//Changes to the origin constraint do not affect the copy of the constraint in the instance of the DynamicConstraint_Container.
//For this reason, the container is being refreshed here							
fbDynConstraintContainer.Clear();
fbDynConstraintContainer.AddConstraint(fbDynConstraintPath);
fbDynConstraintContainer.AddConstraint(fbDynConstraintCoordinates);
END_METHOD

METHOD SetDynConstraint_C : BOOL //Dynamic constraints for individual coordinates.
VAR_INPUT
    V : MC_LREAL; //equivalent to data type LREAL + MC_DEFAULT, MC_MAXIMUM
    A : MC_LREAL; //equivalent to data type LREAL + MC_DEFAULT, MC_MAXIMUM
    D : MC_LREAL; //equivalent to data type LREAL + MC_DEFAULT, MC_MAXIMUM
    J : MC_LREAL; //equivalent to data type LREAL + MC_DEFAULT, MC_MAXIMUM
END_VAR
THIS^.fbDynConstraintCoordinates.SetLimit(	Coordinate := Coord_Mcs_C1, 
											V := V, 
											A := A, 
											D := D, 
											J := J);											

//Changes to the origin constraint do not affect the copy of the constraint in the instance of the DynamicConstraint_Container.
//For this reason, the container is being refreshed here							
fbDynConstraintContainer.Clear();
fbDynConstraintContainer.AddConstraint(fbDynConstraintPath);
fbDynConstraintContainer.AddConstraint(fbDynConstraintCoordinates);
END_METHOD

METHOD SetDynConstraint_Path : BOOL //One dimensional dynamic constraint along the XY-components of a path, ignoring non-tangential effects.
VAR_INPUT
    V : MC_LREAL; //equivalent to data type LREAL + MC_DEFAULT, MC_MAXIMUM
    A : MC_LREAL; //equivalent to data type LREAL + MC_DEFAULT, MC_MAXIMUM
    D : MC_LREAL; //equivalent to data type LREAL + MC_DEFAULT, MC_MAXIMUM
    J : MC_LREAL; //equivalent to data type LREAL + MC_DEFAULT, MC_MAXIMUM
END_VAR
THIS^.fbDynConstraintPath.SetValuesVADJ(V := V, 
										A := A, 
										D := D, 
										J := J);											

//Changes to the origin constraint do not affect the copy of the constraint in the instance of the DynamicConstraint_Container.
//For this reason, the container is being refreshed here							
fbDynConstraintContainer.Clear();
fbDynConstraintContainer.AddConstraint(fbDynConstraintPath);
fbDynConstraintContainer.AddConstraint(fbDynConstraintCoordinates);
END_METHOD

METHOD SetDynConstraint_X : BOOL //Dynamic constraints for individual coordinates.
VAR_INPUT
    V : MC_LREAL; //equivalent to data type LREAL + MC_DEFAULT, MC_MAXIMUM
    A : MC_LREAL; //equivalent to data type LREAL + MC_DEFAULT, MC_MAXIMUM
    D : MC_LREAL; //equivalent to data type LREAL + MC_DEFAULT, MC_MAXIMUM
    J : MC_LREAL; //equivalent to data type LREAL + MC_DEFAULT, MC_MAXIMUM
END_VAR
THIS^.fbDynConstraintCoordinates.SetLimit(	Coordinate := Coord_Mcs_X, 
											V := V, 
											A := A, 
											D := D, 
											J := J);											

//Changes to the origin constraint do not affect the copy of the constraint in the instance of the DynamicConstraint_Container.
//For this reason, the container is being refreshed here							
fbDynConstraintContainer.Clear();
fbDynConstraintContainer.AddConstraint(fbDynConstraintPath);
fbDynConstraintContainer.AddConstraint(fbDynConstraintCoordinates);
END_METHOD

METHOD SetDynConstraint_Y : BOOL //Dynamic constraints for individual coordinates.
VAR_INPUT
    V : MC_LREAL; //equivalent to data type LREAL + MC_DEFAULT, MC_MAXIMUM
    A : MC_LREAL; //equivalent to data type LREAL + MC_DEFAULT, MC_MAXIMUM
    D : MC_LREAL; //equivalent to data type LREAL + MC_DEFAULT, MC_MAXIMUM
    J : MC_LREAL; //equivalent to data type LREAL + MC_DEFAULT, MC_MAXIMUM
END_VAR
THIS^.fbDynConstraintCoordinates.SetLimit(	Coordinate := Coord_Mcs_Y, 
											V := V, 
											A := A, 
											D := D, 
											J := J);											

//Changes to the origin constraint do not affect the copy of the constraint in the instance of the DynamicConstraint_Container.
//For this reason, the container is being refreshed here							
fbDynConstraintContainer.Clear();
fbDynConstraintContainer.AddConstraint(fbDynConstraintPath);
fbDynConstraintContainer.AddConstraint(fbDynConstraintCoordinates);
END_METHOD

METHOD SetDynConstraint_Z : BOOL //Dynamic constraints for individual coordinates.
VAR_INPUT
    V : MC_LREAL; //equivalent to data type LREAL + MC_DEFAULT, MC_MAXIMUM
    A : MC_LREAL; //equivalent to data type LREAL + MC_DEFAULT, MC_MAXIMUM
    D : MC_LREAL; //equivalent to data type LREAL + MC_DEFAULT, MC_MAXIMUM
    J : MC_LREAL; //equivalent to data type LREAL + MC_DEFAULT, MC_MAXIMUM
END_VAR
THIS^.fbDynConstraintCoordinates.SetLimit(	Coordinate := Coord_Mcs_Z, 
											V := MC_DEFAULT, 
											A := A, 
											D := D, 
											J := J);											

//Changes to the origin constraint do not affect the copy of the constraint in the instance of the DynamicConstraint_Container.
//For this reason, the container is being refreshed here							
fbDynConstraintContainer.Clear();
fbDynConstraintContainer.AddConstraint(fbDynConstraintPath);
fbDynConstraintContainer.AddConstraint(fbDynConstraintCoordinates);
END_METHOD

METHOD SetRouteToParent : HRESULT
VAR_INPUT
	ipRoute : I_CH_LIST;
END_VAR
IF ipRoute = 0 THEN
	//Clear on empty input
	THIS^.fbRouteRemaining.Clear();
	THIS^.fbRouteComplete.Clear();
ELSE	
	//set as new route
	THIS^.fbRouteRemaining.Duplicate(ipRoute);
	THIS^.fbRouteComplete.Duplicate(ipRoute);	
END_IF
END_METHOD

{attribute 'monitoring':='call'}
(* Velocity is zero *)
PROPERTY Standstill : BOOL
GET
Standstill := TRUE;
Standstill := Standstill AND THIS^.PlanarMover.MCTOPLC.SET.SetVelo.x = 0;
Standstill := Standstill AND THIS^.PlanarMover.MCTOPLC.SET.SetVelo.y = 0;
Standstill := Standstill AND THIS^.PlanarMover.MCTOPLC.SET.SetVelo.z = 0;
Standstill := Standstill AND THIS^.PlanarMover.MCTOPLC.SET.SetVelo.a = 0;
Standstill := Standstill AND THIS^.PlanarMover.MCTOPLC.SET.SetVelo.b = 0;
Standstill := Standstill AND THIS^.PlanarMover.MCTOPLC.SET.SetVelo.c = 0;
END_GET
END_PROPERTY

METHOD StartExternalSetpoint : HRESULT
THIS^.eActiveCommand 				:= CHALET_NC.E_NcAxisCommands.StartExternalSetpoint;
THIS^.fbFeedback.ActiveCommand 		:= TO_STRING(THIS^.eActiveCommand);		
THIS^.fbFeedback.Busy 				:= TRUE;


IF THIS^.fbMover.MCTOPLC.STD.State <> MC_PLANAR_STATE.Enabled THEN
	//Error wrong state
	
	;//zzz Todo Error message

ELSIF THIS^.bFeedExternalSetpointActive AND THIS^.nSeqStartExternalSetpoint = 999 THEN
	//Do nothing, setpoint is already active	
	THIS^.fbFeedbackExternalSetpointStartSeq.Done		:= TRUE;
	
ELSE
	
	//Start of internal sequence
	THIS^.fbFeedbackExternalSetpointStartSeq.Busy		:= TRUE;
	THIS^.nSeqStartExternalSetpoint := 1;
END_IF



StartExternalSetpoint := S_OK;
END_METHOD

METHOD StopExternalSetpoint : HRESULT
VAR_INPUT
END_VAR
AxisSetpointX.PowerOff();
AxisSetpointY.PowerOff();
AxisSetpointZ.PowerOff();
AxisSetpointA.PowerOff();
AxisSetpointB.PowerOff();
AxisSetpointC.PowerOff();


THIS^.eActiveCommand 				:= CHALET_NC.E_NcAxisCommands.StopExternalSetpoint;
THIS^.fbFeedback.ActiveCommand 		:= TO_STRING(THIS^.eActiveCommand);	
THIS^.fbFeedback.LastCommandAccepted:= TRUE;		


//Reset some flags
THIS^.nSeqStartExternalSetpoint := 0;
THIS^.bEvaluateFeedback := FALSE;
THIS^.ipMasterMover := 0;

IF THIS^.bFeedExternalSetpointActive THEN
	THIS^.fbMover.StopExternalSetpointGeneration(THIS^.fbFeedbackExtStop);	
	THIS^.bFeedExternalSetpointActive 	:= FALSE;
	THIS^.fbFeedback.Busy 				:= TRUE;
ELSE
	THIS^.fbFeedback.Done 				:= TRUE;
END_IF


StopExternalSetpoint := S_OK;
END_METHOD

{attribute 'monitoring':='call'}
//Interface to CHALET system to which this object belongs
PROPERTY System : I_XP_System_PLC
GET
//get I_x_System_PLC interface from I_x_System_Registration
__QUERYINTERFACE(THIS^.ipXpSystem, System);
END_GET
END_PROPERTY

{attribute 'monitoring':='call'}
PROPERTY TargetStation : STRING
GET
TargetStation := THIS^.sTargetStation;
END_GET
SET
THIS^.sTargetStation := TargetStation;
END_SET
END_PROPERTY

METHOD PUBLIC Update : HRESULT
VAR
	ipObject : I_CH_Object;
END_VAR

VAR_INST
	{attribute 'hide'}
	fbCmdNotPossibleCollision : FB_TcAlarm;
	{attribute 'hide'}
	nFeedbackOidOld : UDINT;
	{attribute 'hide'}	
	nOldNcErrorCode 		: UDINT;
	{attribute 'hide'}	
	fbAlarmNcErrorCode		: FB_TcAlarm;
END_VAR
THIS^.Prepare();//Prepare time-critical information, if not already done

THIS^.UpdateExternalSetpoint();
THIS^.UpdateUnknownLevel();

// ********************** Set feedback depending on active command *******************************
CASE THIS^.eActiveCommand OF
	E_NcAxisCommands.None: 
		//Display if a Mover Error is active during no command is active
		IF THIS^.fbMover.Error AND NOT fbFeedback.Error THEN 
			IF THIS^.fbMover.ErrorId <> 1810(*ignore ADSERR_DEVICE_INVALIDSTATE*) THEN
				fbFeedback.ErrorId 			:= THIS^.fbMover.ErrorID;
				fbFeedback.ActiveCommand 	:= TO_STRING(E_NcAxisCommands.None);	
				fbFeedback.ClearObjectInfo();
			END_IF
		END_IF

	E_NcAxisCommands.Initialize:
		fbFeedback.Busy 			:= NOT THIS^.bInitDone;
		fbFeedback.Done 			:= THIS^.bInitDone;
		fbFeedback.ErrorId 			:= 0;
		fbFeedback.ClearObjectInfo();
		                        	
	E_NcAxisCommands.MoveA:     	
		fbFeedback.Busy 			:= fbFeedbackMoveA.Busy;
		fbFeedback.Done 			:= fbFeedbackMoveA.Done;
		fbFeedback.ErrorId 			:= fbFeedbackMoveA.ErrorID;
        fbFeedback.ObjectInfo		:= fbFeedbackMoveA.objectInfo;
                                	
	E_NcAxisCommands.MoveB:     	
		fbFeedback.Busy 			:= fbFeedbackMoveB.Busy;
		fbFeedback.Done 			:= fbFeedbackMoveB.Done;
		fbFeedback.ErrorId 			:= fbFeedbackMoveB.ErrorID;
        fbFeedback.ObjectInfo		:= fbFeedbackMoveB.objectInfo;
                                	
	E_NcAxisCommands.MoveC:     	
		fbFeedback.Busy 			:= fbFeedbackMoveC.Busy;
		fbFeedback.Done 			:= fbFeedbackMoveC.Done;
		fbFeedback.ErrorId 			:= fbFeedbackMoveC.ErrorID;
        fbFeedback.ObjectInfo		:= fbFeedbackMoveC.objectInfo;
                                	
	E_NcAxisCommands.MoveXY:    	
		fbFeedback.Busy 			:= fbFeedbackMoveXY.Busy;
		fbFeedback.Done 			:= fbFeedbackMoveXY.Done;
		fbFeedback.ErrorId 			:= fbFeedbackMoveXY.ErrorID;
        fbFeedback.ObjectInfo		:= fbFeedbackMoveXY.objectInfo;
                                	
	E_NcAxisCommands.MoveZ:     	
		fbFeedback.Busy 			:= fbFeedbackMoveZ.Busy;
		fbFeedback.Done 			:= fbFeedbackMoveZ.Done;
		fbFeedback.ErrorId 			:= fbFeedbackMoveZ.ErrorID;
        fbFeedback.ObjectInfo		:= fbFeedbackMoveZ.objectInfo;
                                	
	E_NcAxisCommands.Enable:    	
		fbFeedback.Busy 			:= fbFeedbackEnable.Busy;
		fbFeedback.Done 			:= fbFeedbackEnable.Done;
		fbFeedback.ErrorId 			:= fbFeedbackEnable.ErrorID;
        fbFeedback.ObjectInfo		:= fbFeedbackEnable.objectInfo;
                                	
	E_NcAxisCommands.Disable:   	
		fbFeedback.Busy 			:= fbFeedbackDisable.Busy;
		fbFeedback.Done 			:= fbFeedbackDisable.Done;
		fbFeedback.ErrorId 			:= fbFeedbackDisable.ErrorID;
        fbFeedback.ObjectInfo		:= fbFeedbackDisable.objectInfo;
                                	
	E_NcAxisCommands.Reset:     	
		fbFeedback.Busy 			:= fbFeedbackReset.Busy;
		fbFeedback.Done 			:= fbFeedbackReset.Done;
		fbFeedback.ErrorId 			:= fbFeedbackReset.ErrorID;
        fbFeedback.ObjectInfo		:= fbFeedbackReset.objectInfo;
                                	
	E_NcAxisCommands.Halt:      	
		fbFeedback.Busy 			:= fbFeedbackHalt.Busy;
		fbFeedback.Done 			:= fbFeedbackHalt.Done;
		fbFeedback.ErrorId 			:= fbFeedbackHalt.ErrorID;
        fbFeedback.ObjectInfo		:= fbFeedbackHalt.objectInfo;

	E_NcAxisCommands.AddToGroupe:
		fbFeedback.Busy 			:= fbFeedbackAddToGrp.Busy;
		fbFeedback.Done 			:= fbFeedbackAddToGrp.Done;
		fbFeedback.ErrorId 			:= fbFeedbackAddToGrp.ErrorID;
        fbFeedback.ObjectInfo		:= fbFeedbackAddToGrp.objectInfo;

	E_NcAxisCommands.RemoveFromGroupe:
		fbFeedback.Busy 			:= fbFeedbackRmvFromGrp.Busy;
		fbFeedback.Done 			:= fbFeedbackRmvFromGrp.Done;
		fbFeedback.ErrorId 			:= fbFeedbackRmvFromGrp.ErrorID;
        fbFeedback.ObjectInfo		:= fbFeedbackRmvFromGrp.objectInfo;
		
	E_NcAxisCommands.JoinTrack:
		fbFeedback.Busy 			:= fbFeedbackJoinTrack.Busy;
		fbFeedback.Done 			:= fbFeedbackJoinTrack.Done;
		fbFeedback.ErrorId 			:= fbFeedbackJoinTrack.ErrorID;
        fbFeedback.ObjectInfo		:= fbFeedbackJoinTrack.objectInfo;
		
	E_NcAxisCommands.MoveOnTrack:
		fbFeedback.Busy 			:= fbFeedbackMoveOnTrack.Busy;
		fbFeedback.Done 			:= fbFeedbackMoveOnTrack.Done;
		fbFeedback.ErrorId 			:= fbFeedbackMoveOnTrack.ErrorID;
        fbFeedback.ObjectInfo		:= fbFeedbackMoveOnTrack.objectInfo;
		
			
	E_NcAxisCommands.StartExternalSetpoint:
		;// in Subroutine "UpdateExternalSetpoint"
	
	E_NcAxisCommands.StopExternalSetpoint:
		;// in Subroutine "UpdateExternalSetpoint"		
			
	E_NcAxisCommands.LiftFromUnknownLevel:
		fbFeedback.Busy 			:= fbFeedbackLiftFromUnknown.Busy;
		fbFeedback.Done 			:= fbFeedbackLiftFromUnknown.Done;
		fbFeedback.ErrorId 			:= fbFeedbackLiftFromUnknown.ErrorID;
        fbFeedback.ClearObjectInfo();
	
	E_NcAxisCommands.LowerToUnknownLevel:
		fbFeedback.Busy 			:= fbFeedbackLowerToUnknown.Busy;
		fbFeedback.Done 			:= fbFeedbackLowerToUnknown.Done;
		fbFeedback.ErrorId 			:= fbFeedbackLowerToUnknown.ErrorID;
        fbFeedback.ClearObjectInfo();
		
	ELSE//External command in subclass
		;
END_CASE


// **********************  Stop to execute commands on .done or .error ***************************
IF fbFeedback.Done OR THIS^.fbFeedback.Error THEN
	eActiveCommand 				:= E_NcAxisCommands.None;
END_IF


// **********************  Get interface to Feedback.ObjectInfo ***************************
IF Feedback.ObjectInfoEx.Id <> 0 AND Feedback.ObjectInfoEx.Id <> nFeedbackOidOld THEN
	CASE Feedback.ObjectInfo.ObjectType OF
		EPlanarObjectType.Mover:
			Feedback.ObjectInfoEx.ipObject := THIS^.ipXPSystem.MoversPresent.FindOID(Feedback.ObjectInfo.Id);
			
		EPlanarObjectType.Track:
				Feedback.ObjectInfoEx.ipObject := THIS^.ipXPSystem.Tracks.FindOID(Feedback.ObjectInfo.Id);
		
		EPlanarObjectType.Environment:
				Feedback.ObjectInfoEx.ipObject := THIS^.ipXPSystem.Enviroment;
				
		ELSE 
			Feedback.ObjectInfoEx.ipObject := 0;
	END_CASE
END_IF
nFeedbackOidOld := Feedback.ObjectInfo.Id;



// **********************  Write NC-Error(Mover.MCTOPLC.ErrorCode) in TC3 Eventlogger ***************************
IF (THIS^.fbMover.MCTOPLC.STD.ErrorCode = 0 AND fbAlarmNcErrorCode.bRaised) THEN
	//No error - Reset	
	fbAlarmNcErrorCode.Clear(0,0);
	
ELSIF (THIS^.fbMover.MCTOPLC.STD.ErrorCode = 0) THEN
	; //Nothing
	
ELSIF (nOldNcErrorCode <> THIS^.fbMover.MCTOPLC.STD.ErrorCode) THEN
	//New Error - Reset, Create and Raise
	fbAlarmNcErrorCode.Clear(0,0);
	fbAlarmNcErrorCode.Create(	eventClass		:= TC_EVENT_CLASSES.Tc3_NcErrorCodes, 
								nEventId		:= (TO_DWORD(THIS^.fbMover.MCTOPLC.STD.ErrorCode) AND 16#FFFF), //Cut HRESULT to 4 digit error code
								eSeverity		:= TcEventSeverity.Error, 
								ipSourceInfo 	:= THIS^.fbSourceInfo, 
								bWithConfirmation := FALSE);
	fbAlarmNcErrorCode.ipArguments.Clear();
	fbAlarmNcErrorCode.Raise(0);
ELSE
	//Alarm is already active
	;
END_IF
nOldNcErrorCode := THIS^.fbMover.MCTOPLC.STD.ErrorCode;



// **********************  Raise alarm on collision error ***************************
ipObject := THIS^.fbFeedback.ObjectInfoEx.ipObject;
IF THIS^.fbFeedback.Error AND (ipObject <> 0) AND NOT fbCmdNotPossibleCollision.bRaised THEN
	fbCmdNotPossibleCollision.CreateEx(stEventEntry := TC_EVENTS.CHALET_XPlanar_Events.CommandNotPossibleCollision, bWithConfirmation := FALSE, ipSourceInfo := THIS^.fbSourceInfo);
	//Command "{1}" not possible. Possible collision with "{2}"
	fbCmdNotPossibleCollision.ipArguments.AddStringByValue(THIS^.fbFeedback.ActiveCommand).AddStringByValue(ipObject.LUID);
	fbCmdNotPossibleCollision.Raise(0);
ELSIF NOT THIS^.fbFeedback.Error OR ipObject = 0 THEN
	fbCmdNotPossibleCollision.Clear(0,0);	
END_IF




//Update xplanar object
THIS^.fbMover.Update();



//Update feedback object
fbFeedbackMoveA.Update(); 
fbFeedbackMoveB.Update(); 
fbFeedbackMoveC.Update(); 
fbFeedbackMoveXY.Update(); 
fbFeedbackMoveZ.Update(); 
fbFeedbackEnable.Update(); 
fbFeedbackDisable.Update(); 
fbFeedbackReset.Update(); 
fbFeedbackAddToGrp.Update(); 
fbFeedbackRmvFromGrp.Update(); 
fbFeedbackHalt.Update(); 
fbFeedbackJoinTrack.Update(); 
fbFeedbackMoveOnTrack.Update();
END_METHOD

METHOD PROTECTED UpdateExternalSetpoint : HRESULT
VAR
	SetPos, SetVelo, SetAcc : MoverVector;
	hr : HRESULT;
	stStartOptions : ST_ExternalSetpointGenerationOptions;
	stPosDifferenceToMasterMover : MoverVector;
	stPosOffsetMasterMover : MoverVector;
	stVeloOffsetMasterMover : MoverVector;
	stAccOffsetMasterMover : MoverVector;
END_VAR
IF NOT THIS^.Enabled THEN
	THIS^.nSeqStartExternalSetpoint := 0;
	THIS^.bFeedExternalSetpointActive := FALSE;
	THIS^.bEvaluateFeedback := FALSE;
END_IF


CASE nSeqStartExternalSetpoint OF
	0: //Wait for start
		;
		
	1: 	//store position of Master-Mover
		IF (THIS^.ipMasterMover <> 0) THEN
			THIS^.stMasterPositionAtStart := THIS^.ipMasterMover.PositionSet;
		END_IF

		//Reset all axis
		IF AxisSetpointX.Mapped THEN
			AxisSetpointX.Reset();
		END_IF
		IF AxisSetpointY.Mapped THEN
			AxisSetpointY.Reset();
		END_IF
		IF AxisSetpointZ.Mapped THEN
			AxisSetpointZ.Reset();
		END_IF
		IF AxisSetpointA.Mapped THEN
			AxisSetpointA.Reset();
		END_IF
		IF AxisSetpointB.Mapped THEN
			AxisSetpointB.Reset();
		END_IF
		IF AxisSetpointC.Mapped THEN
			AxisSetpointC.Reset();
		END_IF
		nSeqStartExternalSetpoint := nSeqStartExternalSetpoint + 1;		
		
		
	2: //Wait for feedback
		IF AxisSetpointX.Mapped THEN hr := GetMostSignificant(hr, AxisSetpointX.Feedback.HR); END_IF
		IF AxisSetpointY.Mapped THEN hr := GetMostSignificant(hr, AxisSetpointY.Feedback.HR); END_IF
		IF AxisSetpointZ.Mapped THEN hr := GetMostSignificant(hr, AxisSetpointZ.Feedback.HR); END_IF
		IF AxisSetpointA.Mapped THEN hr := GetMostSignificant(hr, AxisSetpointA.Feedback.HR); END_IF
		IF AxisSetpointB.Mapped THEN hr := GetMostSignificant(hr, AxisSetpointB.Feedback.HR); END_IF
		IF AxisSetpointC.Mapped THEN hr := GetMostSignificant(hr, AxisSetpointC.Feedback.HR); END_IF	
		IF hr = S_OK THEN
		 	nSeqStartExternalSetpoint := nSeqStartExternalSetpoint + 1;	
		END_IF
		
	3: 	//Reset all axis
		IF AxisSetpointX.Mapped THEN
			AxisSetpointX.PowerOn();
		END_IF
		IF AxisSetpointY.Mapped THEN
			AxisSetpointY.PowerOn();
		END_IF
		IF AxisSetpointZ.Mapped THEN
			AxisSetpointZ.PowerOn();
		END_IF
		IF AxisSetpointA.Mapped THEN
			AxisSetpointA.PowerOn();
		END_IF
		IF AxisSetpointB.Mapped THEN
			AxisSetpointB.PowerOn();
		END_IF
		IF AxisSetpointC.Mapped THEN
			AxisSetpointC.PowerOn();
		END_IF
		nSeqStartExternalSetpoint := nSeqStartExternalSetpoint + 1;		
		
	4: //Wait for feedback
		IF AxisSetpointX.Mapped THEN hr := GetMostSignificant(hr, AxisSetpointX.Feedback.HR); END_IF
		IF AxisSetpointY.Mapped THEN hr := GetMostSignificant(hr, AxisSetpointY.Feedback.HR); END_IF
		IF AxisSetpointZ.Mapped THEN hr := GetMostSignificant(hr, AxisSetpointZ.Feedback.HR); END_IF
		IF AxisSetpointA.Mapped THEN hr := GetMostSignificant(hr, AxisSetpointA.Feedback.HR); END_IF
		IF AxisSetpointB.Mapped THEN hr := GetMostSignificant(hr, AxisSetpointB.Feedback.HR); END_IF
		IF AxisSetpointC.Mapped THEN hr := GetMostSignificant(hr, AxisSetpointC.Feedback.HR); END_IF	
		IF hr = S_OK THEN
		 	nSeqStartExternalSetpoint := nSeqStartExternalSetpoint + 1;	
		END_IF

	5: 	//Enable all axis
		IF AxisSetpointX.Mapped THEN
			AxisSetpointX.SetActPosition(0.0);
		END_IF
		IF AxisSetpointY.Mapped THEN
			AxisSetpointY.SetActPosition(0.0);
		END_IF
		IF AxisSetpointZ.Mapped THEN
			AxisSetpointZ.SetActPosition(0.0);
		END_IF
		IF AxisSetpointA.Mapped THEN
			AxisSetpointA.SetActPosition(0.0);
		END_IF
		IF AxisSetpointB.Mapped THEN
			AxisSetpointB.SetActPosition(0.0);
		END_IF
		IF AxisSetpointC.Mapped THEN
			AxisSetpointC.SetActPosition(0.0);
		END_IF
		nSeqStartExternalSetpoint := nSeqStartExternalSetpoint + 1;		
		
	6: //Wait for feedback
		IF AxisSetpointX.Mapped THEN hr := GetMostSignificant(hr, AxisSetpointX.Feedback.HR); END_IF
		IF AxisSetpointY.Mapped THEN hr := GetMostSignificant(hr, AxisSetpointY.Feedback.HR); END_IF
		IF AxisSetpointZ.Mapped THEN hr := GetMostSignificant(hr, AxisSetpointZ.Feedback.HR); END_IF
		IF AxisSetpointA.Mapped THEN hr := GetMostSignificant(hr, AxisSetpointA.Feedback.HR); END_IF
		IF AxisSetpointB.Mapped THEN hr := GetMostSignificant(hr, AxisSetpointB.Feedback.HR); END_IF
		IF AxisSetpointC.Mapped THEN hr := GetMostSignificant(hr, AxisSetpointC.Feedback.HR); END_IF	
		IF hr = S_OK THEN
		 	nSeqStartExternalSetpoint := nSeqStartExternalSetpoint + 1;	
		END_IF

		
	7: // Activate external setpoint mode on mover
		stStartOptions.Mode := MC_EXTERNAL_SET_POSITION_MODE.Relative;
		THIS^.fbMover.StartExternalSetpointGeneration(	commandFeedback	:= THIS^.fbFeedbackExtStart,
														options 		:= stStartOptions);
		THIS^.bFeedExternalSetpointActive := TRUE;												
		nSeqStartExternalSetpoint := nSeqStartExternalSetpoint + 1;
	
		
	8: 
		THIS^.bEvaluateFeedback := TRUE;
		IF THIS^.fbFeedbackExtStart.Done THEN
			//Finish Sequence
			fbFeedbackExternalSetpointStartSeq.Done := TRUE;
			nSeqStartExternalSetpoint := 999;
		END_IF
		
	999: // finish seqence feedback
		
		
	1000..1999:
		//Error
		fbFeedbackExternalSetpointStartSeq.HR := E_FAIL;
END_CASE



IF THIS^.bFeedExternalSetpointActive THEN
	SetPos.X := AxisSetpointX.SetPosition;
	SetPos.Y := AxisSetpointY.SetPosition;
	SetPos.Z := AxisSetpointZ.SetPosition;
	SetPos.A := AxisSetpointA.SetPosition;
	SetPos.B := AxisSetpointB.SetPosition;
	SetPos.C := AxisSetpointC.SetPosition;
	
	SetVelo.X := AxisSetpointX.SetVelocity;
	SetVelo.Y := AxisSetpointY.SetVelocity;
	SetVelo.Z := AxisSetpointZ.SetVelocity;
	SetVelo.A := AxisSetpointA.SetVelocity;
	SetVelo.B := AxisSetpointB.SetVelocity;
	SetVelo.C := AxisSetpointC.SetVelocity;
	
	SetAcc.X := AxisSetpointX.SetAcceleration;
	SetAcc.Y := AxisSetpointY.SetAcceleration;
	SetAcc.Z := AxisSetpointZ.SetAcceleration;
	SetAcc.A := AxisSetpointA.SetAcceleration;
	SetAcc.B := AxisSetpointB.SetAcceleration;
	SetAcc.C := AxisSetpointC.SetAcceleration;
	
	IF THIS^.ipMasterMover <> 0 THEN
		//Difference to gearIn position
		stPosDifferenceToMasterMover := F_Vector_Subtraction(	minuend := THIS^.ipMasterMover.PositionSet, 
																subtrahend := stMasterPositionAtStart);
		//Add scaling factor	
		stPosOffsetMasterMover := F_Vector_Multiplication(	factor1 := stPosDifferenceToMasterMover,
															factor2 := THIS^.stMasterMovementScaling);							
		stVeloOffsetMasterMover := F_Vector_Multiplication(	factor1 := THIS^.ipMasterMover.VelocitySet,
															factor2 := THIS^.stMasterMovementScaling);							
		stAccOffsetMasterMover := F_Vector_Multiplication(	factor1 := THIS^.ipMasterMover.AccelerationSet,
															factor2 := THIS^.stMasterMovementScaling);						
		
		
		//Add Mastermover-Offest to 6-Axis-Offset
		SetPos := F_Vector_Addition( 	summand1 := stPosOffsetMasterMover,
									 	summand2 := SetPos);
		SetVelo := F_Vector_Addition( 	summand1 := stVeloOffsetMasterMover,
									 	summand2 := SetVelo);
		SetAcc := F_Vector_Addition( 	summand1 := stAccOffsetMasterMover,
									 	summand2 := SetAcc);
														
	END_IF
	
	//Send data to mover
	THIS^.fbMover.SetExternalSetpoint(	setPosition 		:= SetPos, 
										setVelocity 		:= SetVelo,
										setAcceleration 	:= SetAcc);
END_IF



CASE THIS^.eActiveCommand OF
	//Add the 6 axis to the feedback			
	E_NcAxisCommands.StartExternalSetpoint:
		//Only check MC_PlanarFeedback if cmd is active. Ignore old feedback
		IF THIS^.bEvaluateFeedback THEN
			fbFeedback.Busy 		:= fbFeedbackExtStart.Busy;
			fbFeedback.Done 		:= fbFeedbackExtStart.Done;
			fbFeedback.ErrorId 		:= fbFeedbackExtStart.ErrorID;
			fbFeedback.ClearObjectInfo();
		END_IF
		fbFeedback.HR := GetMostSignificant(fbFeedback.HR, fbFeedbackExternalSetpointStartSeq.HR);
		IF AxisSetpointX.Mapped THEN fbFeedback.HR := GetMostSignificant(fbFeedback.HR, AxisSetpointX.Feedback.HR);END_IF
		IF AxisSetpointY.Mapped THEN fbFeedback.HR := GetMostSignificant(fbFeedback.HR, AxisSetpointY.Feedback.HR);END_IF
		IF AxisSetpointZ.Mapped THEN fbFeedback.HR := GetMostSignificant(fbFeedback.HR, AxisSetpointZ.Feedback.HR);END_IF
		IF AxisSetpointA.Mapped THEN fbFeedback.HR := GetMostSignificant(fbFeedback.HR, AxisSetpointA.Feedback.HR);END_IF
		IF AxisSetpointB.Mapped THEN fbFeedback.HR := GetMostSignificant(fbFeedback.HR, AxisSetpointB.Feedback.HR);END_IF
		IF AxisSetpointC.Mapped THEN fbFeedback.HR := GetMostSignificant(fbFeedback.HR, AxisSetpointC.Feedback.HR);END_IF
		
	//Add the 6 axis to the feedback	
	E_NcAxisCommands.StopExternalSetpoint:
		fbFeedback.Busy 		:= fbFeedbackExtStop.Busy;
		fbFeedback.Done 		:= fbFeedbackExtStop.Done;
		fbFeedback.ErrorId 		:= fbFeedbackExtStop.ErrorID;
		fbFeedback.ClearObjectInfo(); 
		IF AxisSetpointX.Mapped THEN fbFeedback.HR := GetMostSignificant(fbFeedback.HR, AxisSetpointX.Feedback.HR);END_IF
		IF AxisSetpointY.Mapped THEN fbFeedback.HR := GetMostSignificant(fbFeedback.HR, AxisSetpointY.Feedback.HR);END_IF
		IF AxisSetpointZ.Mapped THEN fbFeedback.HR := GetMostSignificant(fbFeedback.HR, AxisSetpointZ.Feedback.HR);END_IF
		IF AxisSetpointA.Mapped THEN fbFeedback.HR := GetMostSignificant(fbFeedback.HR, AxisSetpointA.Feedback.HR);END_IF
		IF AxisSetpointB.Mapped THEN fbFeedback.HR := GetMostSignificant(fbFeedback.HR, AxisSetpointB.Feedback.HR);END_IF
		IF AxisSetpointC.Mapped THEN fbFeedback.HR := GetMostSignificant(fbFeedback.HR, AxisSetpointC.Feedback.HR);END_IF
END_CASE		


fbFeedbackExtStart.Update(); 
fbFeedbackExtStop.Update(); 


IF AxisSetpointX.Mapped THEN AxisSetpointX.Update() ;END_IF
IF AxisSetpointY.Mapped THEN AxisSetpointY.Update() ;END_IF
IF AxisSetpointZ.Mapped THEN AxisSetpointZ.Update() ;END_IF
IF AxisSetpointA.Mapped THEN AxisSetpointA.Update() ;END_IF
IF AxisSetpointB.Mapped THEN AxisSetpointB.Update() ;END_IF
IF AxisSetpointC.Mapped THEN AxisSetpointC.Update() ;END_IF
END_METHOD

METHOD PROTECTED UpdateUnknownLevel : HRESULT
VAR
	hr : HRESULT;
	stForceLimitMax: Tc3_XPlanarUtility.Force6D;
	stForceLimitMin: Tc3_XPlanarUtility.Force6D;
	stPosLagValueTemp : MoverVector;
	ipComObject: Tc3_Module.ITComObject;
	pstForcesAtBeginn : POINTER TO MoverVector;
END_VAR
VAR_INST
	fLowerNPerS : LREAL := 30.0;
	fLiftNPerS : LREAL := 50.0;
	fMaxForceFactor : LREAL := 1.0;
	fMinForceFactor : LREAL := 0.1;
	fPowerFactor : LREAL := 1.0;
	fCycleTime_s : LREAL; //[s]	
	bDoOnceIfDisabled : BOOL;
	stLagValuesAtBeginn : MoverVector;
	stForcesAtBeginn :  MoverVector;
	stForceLimitMaxAtBeginn : Tc3_XPlanarUtility.Force6D;
	stForceLimitMinAtBeginn : Tc3_XPlanarUtility.Force6D;
	stValideMinForce		: Tc3_XPlanarUtility.Force6D;
END_VAR
VAR CONSTANT
	N_PTCID_ForceLimitMax : PTCID := 16#03175051;
	N_PTCID_ForceLimitMin : PTCID := 16#03175052;
END_VAR
IF NOT THIS^.Enabled THEN
	THIS^.nSeqLowerToUnknown := 0;
	THIS^.nSeqLiftFromUnknown := 0;
	
	fCycleTime_s :=  TO_LREAL(TwinCAT_SystemInfoVarList._TaskInfo[THIS^.nTaskIndex].CycleTime(*100ns*)) / 10_000_000.0;
	stLagValuesAtBeginn := THIS^.UtilityMcMover.GetMaximumPositionLagValue();
END_IF

//if no TcIoMover is linked e.g. MC-Mover is in Simulation Mover:
IF THIS^.UtilityTcIoMover = 0 THEN
	IF fbFeedbackLowerToUnknown.Busy THEN
		fbFeedbackLowerToUnknown.Done := TRUE;
	END_IF
	IF fbFeedbackLiftFromUnknown.Busy THEN
		fbFeedbackLiftFromUnknown.Done := TRUE;
	END_IF
	RETURN;
END_IF



IF THIS^.ipXpSystem.Disabled AND bDoOnceIfDisabled THEN
	bDoOnceIfDisabled := FALSE;
	fPowerFactor := fMaxForceFactor;
	
	FW_ObjMgr_GetObjectInstance(oid:= THIS^.UtilityTcIoMover.ObjectId, iid:= TC_GLOBAL_IID_LIST.IID_ITComObject, pipUnk:= ADR(ipComObject));
	IF ipComObject <> 0 THEN
		// No minimum can be set if one of the 6 values in the struct is greater than the maximum. Equal is allowed.
		// The minimum is therefore first written to something valid. Followed by Max and the original minimum
		hr := ipComObject.TcSetObjPara(pid := N_PTCID_ForceLimitMin, nData := SIZEOF(stValideMinForce), pData := ADR(stValideMinForce), pgp := 0);
		hr := ipComObject.TcSetObjPara(pid := N_PTCID_ForceLimitMax, nData := SIZEOF(stForceLimitMaxAtBeginn), pData := ADR(stForceLimitMaxAtBeginn), pgp := 0);
		hr := ipComObject.TcSetObjPara(pid := N_PTCID_ForceLimitMin, nData := SIZEOF(stForceLimitMinAtBeginn), pData := ADR(stForceLimitMinAtBeginn), pgp := 0);
		FW_SafeRelease(ADR(ipComObject));
	END_IF

	THIS^.UtilityMcMover.SetMaximumPositionLagValue(stLagValuesAtBeginn);
END_IF


//Down
CASE nSeqLowerToUnknown OF
	0: //Wait for start
		;
		
	1: // Check if not already lewered	
		IF fPowerFactor = fMinForceFactor THEN
			nSeqLowerToUnknown := 999;
		ELSE
			nSeqLowerToUnknown := 5;
		END_IF
		
	5:	//Get some values
		pstForcesAtBeginn := THIS^.UtilityTcIoMover.ScopeAdr.GetOutputForce();
		stForcesAtBeginn := pstForcesAtBeginn^;
		stForceLimitMaxAtBeginn := THIS^.UtilityTcIoMover.GetForceLimitMax();
		stForceLimitMinAtBeginn := THIS^.UtilityTcIoMover.GetForceLimitMin();
		stValideMinForce.Fx := (stForceLimitMinAtBeginn.Fx * fMinForceFactor);
		stValideMinForce.Fy := (stForceLimitMinAtBeginn.Fy * fMinForceFactor);
		stValideMinForce.Fz := (stForceLimitMinAtBeginn.Fz * fMinForceFactor);
		stValideMinForce.Mx := (stForceLimitMinAtBeginn.Mx * fMinForceFactor);
		stValideMinForce.My := (stForceLimitMinAtBeginn.My * fMinForceFactor);
		stValideMinForce.Mz := (stForceLimitMinAtBeginn.Mz * fMinForceFactor);
		bDoOnceIfDisabled := TRUE;
		
		stPosLagValueTemp := stLagValuesAtBeginn;
		stPosLagValueTemp.z := THIS^.PositionSet.z + 0.5;
		THIS^.UtilityMcMover.SetMaximumPositionLagValue(stPosLagValueTemp);
		
		
		//0.0 - 1.0
		fPowerFactor := (stForcesAtBeginn.z / stForceLimitMaxAtBeginn.Fz);
		
		//add 5%
		fPowerFactor := fPowerFactor + 0.05;
		
		//Limit to 0.1 - 1.0
		fPowerFactor := MIN(fPowerFactor, fMaxForceFactor);
		fPowerFactor := MAX(fPowerFactor, fMinForceFactor);
		
		//set force Z, a and b
		stForceLimitMin := stForceLimitMinAtBeginn;		
		stForceLimitMin.fz := stForceLimitMin.Fz * fPowerFactor;
		stForceLimitMin.Mx := stForceLimitMin.Mx * fPowerFactor;
		stForceLimitMin.My := stForceLimitMin.My * fPowerFactor;
		
		stForceLimitMax := stForceLimitMaxAtBeginn;	
		stForceLimitMax.fz := stForceLimitMax.Fz * fPowerFactor;
		stForceLimitMax.Mx := stForceLimitMax.Mx * fPowerFactor;
		stForceLimitMax.My := stForceLimitMax.My * fPowerFactor;

		// 13.01.2025 Todo PLC Chash if Min > Max. use objParm insted
		//	THIS^.TcIoXPlanarMover.SetForceLimitMin(stForceLimitMin);
		//	THIS^.TcIoXPlanarMover.SetForceLimitMax(stForceLimitMax);
		FW_ObjMgr_GetObjectInstance(oid:= THIS^.UtilityTcIoMover.ObjectId, iid:= TC_GLOBAL_IID_LIST.IID_ITComObject, pipUnk:= ADR(ipComObject));
		IF ipComObject <> 0 THEN	
			// No minimum can be set if one of the 6 values in the struct is greater than the maximum. Equal is allowed.
			// The minimum is therefore first written to something valid. Followed by Max and the original minimum
			hr := ipComObject.TcSetObjPara(pid := N_PTCID_ForceLimitMin, nData := SIZEOF(stValideMinForce), pData := ADR(stValideMinForce), pgp := 0);
			hr := ipComObject.TcSetObjPara(pid := N_PTCID_ForceLimitMax, nData := SIZEOF(stForceLimitMax), pData := ADR(stForceLimitMax), pgp := 0);
			hr := ipComObject.TcSetObjPara(pid := N_PTCID_ForceLimitMin, nData := SIZEOF(stForceLimitMin), pData := ADR(stForceLimitMin), pgp := 0);
			FW_SafeRelease(ADR(ipComObject));
		END_IF

	
		nSeqLowerToUnknown := 10;
		
		
	10: 	
		//A lowering of the mover was detected followed by speed ~0
		IF (THIS^.PositionAct.z < THIS^.PositionSet.z * 0.5) AND (ABS(THIS^.VelocityAct.z) < 5.0)  THEN
			nSeqLowerToUnknown := 20;
			
		ELSIF (fPowerFactor <= fMinForceFactor) THEN
			nSeqLowerToUnknown := 20;
				
		ELSE
			//Reduce force each cycle
			fPowerFactor := fPowerFactor - ((fLowerNPerS/stForceLimitMaxAtBeginn.Fz) * fCycleTime_s);
					
			//Limit to 0.1 - 1.0
			fPowerFactor := MIN(fPowerFactor, fMaxForceFactor);
			fPowerFactor := MAX(fPowerFactor, fMinForceFactor);
			
			//set force Z, a and b to current + 10%
			stForceLimitMin := stForceLimitMinAtBeginn;		
			stForceLimitMin.fz := stForceLimitMin.Fz * fPowerFactor;
			stForceLimitMin.Mx := stForceLimitMin.Mx * fPowerFactor;
			stForceLimitMin.My := stForceLimitMin.My * fPowerFactor;
			
			stForceLimitMax := stForceLimitMaxAtBeginn;	
			stForceLimitMax.fz := stForceLimitMax.Fz * fPowerFactor;
			stForceLimitMax.Mx := stForceLimitMax.Mx * fPowerFactor;
			stForceLimitMax.My := stForceLimitMax.My * fPowerFactor;
	
			// 13.01.2025 Todo PLC Chash if Min > Max. use objParm insted
			//	THIS^.TcIoXPlanarMover.SetForceLimitMin(stForceLimitMin);
			//	THIS^.TcIoXPlanarMover.SetForceLimitMax(stForceLimitMax);
			FW_ObjMgr_GetObjectInstance(oid:= THIS^.UtilityTcIoMover.ObjectId, iid:= TC_GLOBAL_IID_LIST.IID_ITComObject, pipUnk:= ADR(ipComObject));
			IF ipComObject <> 0 THEN
				// No minimum can be set if one of the 6 values in the struct is greater than the maximum. Equal is allowed.
				// The minimum is therefore first written to something valid. Followed by Max and the original minimum
				hr := ipComObject.TcSetObjPara(pid := N_PTCID_ForceLimitMin, nData := SIZEOF(stValideMinForce), pData := ADR(stValideMinForce), pgp := 0);
				hr := ipComObject.TcSetObjPara(pid := N_PTCID_ForceLimitMax, nData := SIZEOF(stForceLimitMax), pData := ADR(stForceLimitMax), pgp := 0);
				hr := ipComObject.TcSetObjPara(pid := N_PTCID_ForceLimitMin, nData := SIZEOF(stForceLimitMin), pData := ADR(stForceLimitMin), pgp := 0);
				FW_SafeRelease(ADR(ipComObject));
			END_IF

	
		END_IF
	
		
	20: // Reduce Force to minimum
		fPowerFactor := fMinForceFactor;
		
		//set force Z, a and b to minimum
		stForceLimitMin := stForceLimitMinAtBeginn;		
		stForceLimitMin.fz := stForceLimitMin.Fz * fPowerFactor;
		stForceLimitMin.Mx := stForceLimitMin.Mx * fPowerFactor;
		stForceLimitMin.My := stForceLimitMin.My * fPowerFactor;
		
		stForceLimitMax := stForceLimitMaxAtBeginn;	
		stForceLimitMax.fz := stForceLimitMax.Fz * fPowerFactor;
		stForceLimitMax.Mx := stForceLimitMax.Mx * fPowerFactor;
		stForceLimitMax.My := stForceLimitMax.My * fPowerFactor;
	    
	    
		// 13.01.2025 Todo PLC Chash if Min > Max. use objParm insted
		//	THIS^.TcIoXPlanarMover.SetForceLimitMin(stForceLimitMin);
		//	THIS^.TcIoXPlanarMover.SetForceLimitMax(stForceLimitMax);
		FW_ObjMgr_GetObjectInstance(oid:= THIS^.UtilityTcIoMover.ObjectId, iid:= TC_GLOBAL_IID_LIST.IID_ITComObject, pipUnk:= ADR(ipComObject));
		IF ipComObject <> 0 THEN
			// No minimum can be set if one of the 6 values in the struct is greater than the maximum. Equal is allowed.
			// The minimum is therefore first written to something valid. Followed by Max and the original minimum
			hr := ipComObject.TcSetObjPara(pid := N_PTCID_ForceLimitMin, nData := SIZEOF(stValideMinForce), pData := ADR(stValideMinForce), pgp := 0);
			hr := ipComObject.TcSetObjPara(pid := N_PTCID_ForceLimitMax, nData := SIZEOF(stForceLimitMax), pData := ADR(stForceLimitMax), pgp := 0);
			hr := ipComObject.TcSetObjPara(pid := N_PTCID_ForceLimitMin, nData := SIZEOF(stForceLimitMin), pData := ADR(stForceLimitMin), pgp := 0);
			FW_SafeRelease(ADR(ipComObject));
		END_IF

		
		nSeqLowerToUnknown := 999;
				
	999: // finish seqence feedback
		fbFeedbackLowerToUnknown.Done := TRUE;
		
	1000..1999:
		//Error
		fbFeedbackLowerToUnknown.HR := E_FAIL;
END_CASE



//Up
CASE nSeqLiftFromUnknown OF
	0: //Wait for start
		;
		
	1: // Check if not already lifted	
		IF fPowerFactor = fMaxForceFactor THEN
			nSeqLiftFromUnknown := 999;
		ELSE
			nSeqLiftFromUnknown := 5;
		END_IF		
		
	5: 
		//0.0 - 1.0
		fPowerFactor := (stForcesAtBeginn.z / stForceLimitMaxAtBeginn.Fz);
		
		// -5%
		fPowerFactor := fPowerFactor - 0.05;
		
		//Limit to 0.1 - 1.0
		fPowerFactor := MIN(fPowerFactor, fMaxForceFactor);
		fPowerFactor := MAX(fPowerFactor, fMinForceFactor);
		
		//set force Z, a and b
		stForceLimitMin := stForceLimitMinAtBeginn;		
		stForceLimitMin.fz := stForceLimitMin.Fz * fPowerFactor;
		stForceLimitMin.Mx := stForceLimitMin.Mx * fPowerFactor;
		stForceLimitMin.My := stForceLimitMin.My * fPowerFactor;
		
		stForceLimitMax := stForceLimitMaxAtBeginn;	
		stForceLimitMax.fz := stForceLimitMax.Fz * fPowerFactor;
		stForceLimitMax.Mx := stForceLimitMax.Mx * fPowerFactor;
		stForceLimitMax.My := stForceLimitMax.My * fPowerFactor;

		// 13.01.2025 Todo PLC Chash if Min > Max. use objParm insted
		//THIS^.TcIoXPlanarMover.SetForceLimitMax(stForceLimitMax);
		//THIS^.TcIoXPlanarMover.SetForceLimitMin(stForceLimitMin);
		FW_ObjMgr_GetObjectInstance(oid:= THIS^.UtilityTcIoMover.ObjectId, iid:= TC_GLOBAL_IID_LIST.IID_ITComObject, pipUnk:= ADR(ipComObject));
		IF ipComObject <> 0 THEN
			// No minimum can be set if one of the 6 values in the struct is greater than the maximum. Equal is allowed.
			// The minimum is therefore first written to something valid. Followed by Max and the original minimum
			hr := ipComObject.TcSetObjPara(pid := N_PTCID_ForceLimitMin, nData := SIZEOF(stValideMinForce), pData := ADR(stValideMinForce), pgp := 0);
			hr := ipComObject.TcSetObjPara(pid := N_PTCID_ForceLimitMax, nData := SIZEOF(stForceLimitMax), pData := ADR(stForceLimitMax), pgp := 0);
			hr := ipComObject.TcSetObjPara(pid := N_PTCID_ForceLimitMin, nData := SIZEOF(stForceLimitMin), pData := ADR(stForceLimitMin), pgp := 0);
			FW_SafeRelease(ADR(ipComObject));
		END_IF
		
		nSeqLiftFromUnknown := 10;
		

		
	10: 	
		//A lift of the mover was detected followed by speed ~0
		IF (THIS^.PositionAct.z > THIS^.PositionSet.z * 0.5) AND (ABS(THIS^.VelocityAct.z) < 5.0)  THEN
			nSeqLiftFromUnknown := 20;
			
		ELSIF (fPowerFactor >= fMaxForceFactor ) THEN
			nSeqLiftFromUnknown := 20;
				
		ELSE
			//Reduce force each cycle
			fPowerFactor := fPowerFactor + ((fLiftNPerS/stForceLimitMaxAtBeginn.Fz) * fCycleTime_s);
					
			//Limit to 0.1 - 1.0
			fPowerFactor := MIN(fPowerFactor, fMaxForceFactor);
			fPowerFactor := MAX(fPowerFactor, fMinForceFactor);
			
			//set force Z, a and b 
			stForceLimitMin := stForceLimitMinAtBeginn;		
			stForceLimitMin.fz := stForceLimitMin.Fz * fPowerFactor;
			stForceLimitMin.Mx := stForceLimitMin.Mx * fPowerFactor;
			stForceLimitMin.My := stForceLimitMin.My * fPowerFactor;
			
			stForceLimitMax := stForceLimitMaxAtBeginn;	
			stForceLimitMax.fz := stForceLimitMax.Fz * fPowerFactor;
			stForceLimitMax.Mx := stForceLimitMax.Mx * fPowerFactor;
			stForceLimitMax.My := stForceLimitMax.My * fPowerFactor;
	
	
		// 13.01.2025 Todo PLC Chash if Min > Max. use objParm insted
		//THIS^.TcIoXPlanarMover.SetForceLimitMax(stForceLimitMax);
		//THIS^.TcIoXPlanarMover.SetForceLimitMin(stForceLimitMin);
		FW_ObjMgr_GetObjectInstance(oid:= THIS^.UtilityTcIoMover.ObjectId, iid:= TC_GLOBAL_IID_LIST.IID_ITComObject, pipUnk:= ADR(ipComObject));
		IF ipComObject <> 0 THEN
			// No minimum can be set if one of the 6 values in the struct is greater than the maximum. Equal is allowed.
			// The minimum is therefore first written to something valid. Followed by Max and the original minimum
			hr := ipComObject.TcSetObjPara(pid := N_PTCID_ForceLimitMin, nData := SIZEOF(stValideMinForce), pData := ADR(stValideMinForce), pgp := 0);
			hr := ipComObject.TcSetObjPara(pid := N_PTCID_ForceLimitMax, nData := SIZEOF(stForceLimitMax), pData := ADR(stForceLimitMax), pgp := 0);
			hr := ipComObject.TcSetObjPara(pid := N_PTCID_ForceLimitMin, nData := SIZEOF(stForceLimitMin), pData := ADR(stForceLimitMin), pgp := 0);
			FW_SafeRelease(ADR(ipComObject));
		END_IF
	
		END_IF
	
		
	20: // Reduce Force to normal			
		fPowerFactor := fMaxForceFactor;
		
		//set force Z, a and b to minimum
		stForceLimitMin := stForceLimitMinAtBeginn;		
		stForceLimitMin.fz := stForceLimitMin.Fz * fPowerFactor;
		stForceLimitMin.Mx := stForceLimitMin.Mx * fPowerFactor;
		stForceLimitMin.My := stForceLimitMin.My * fPowerFactor;
		
		stForceLimitMax := stForceLimitMaxAtBeginn;	
		stForceLimitMax.fz := stForceLimitMax.Fz * fPowerFactor;
		stForceLimitMax.Mx := stForceLimitMax.Mx * fPowerFactor;
		stForceLimitMax.My := stForceLimitMax.My * fPowerFactor;
	    	
		// 13.01.2025 Todo PLC Chash if Min > Max. use objParm insted
		//THIS^.TcIoXPlanarMover.SetForceLimitMax(stForceLimitMax);
		//THIS^.TcIoXPlanarMover.SetForceLimitMin(stForceLimitMin);
		FW_ObjMgr_GetObjectInstance(oid:= THIS^.UtilityTcIoMover.ObjectId, iid:= TC_GLOBAL_IID_LIST.IID_ITComObject, pipUnk:= ADR(ipComObject));
		IF ipComObject <> 0 THEN
			// No minimum can be set if one of the 6 values in the struct is greater than the maximum. Equal is allowed.
			// The minimum is therefore first written to something valid. Followed by Max and the original minimum
			hr := ipComObject.TcSetObjPara(pid := N_PTCID_ForceLimitMin, nData := SIZEOF(stValideMinForce), pData := ADR(stValideMinForce), pgp := 0);
			hr := ipComObject.TcSetObjPara(pid := N_PTCID_ForceLimitMax, nData := SIZEOF(stForceLimitMax), pData := ADR(stForceLimitMax), pgp := 0);
			hr := ipComObject.TcSetObjPara(pid := N_PTCID_ForceLimitMin, nData := SIZEOF(stForceLimitMin), pData := ADR(stForceLimitMin), pgp := 0);
			FW_SafeRelease(ADR(ipComObject));
		END_IF
		
		
		THIS^.UtilityMcMover.SetMaximumPositionLagValue(stLagValuesAtBeginn);
        
		nSeqLiftFromUnknown := 999;
				
	999: // finish seqence feedback
		fbFeedbackLiftFromUnknown.Done := TRUE;
		
	1000..1999:
		//Error
		fbFeedbackLiftFromUnknown.HR := E_FAIL;
END_CASE
END_METHOD

{attribute 'monitoring':='call'}
PROPERTY UtilityMcMover : Tc3_XPlanarUtility.I_McPlanarMover
GET
UtilityMcMover :=  THIS^.ipMcMover;
END_GET
END_PROPERTY

{attribute 'monitoring':='call'}
PROPERTY UtilityTcIoMover : Tc3_XPlanarUtility.I_TcIoXPlanarMover
GET
VAR
;
END_VAR
UtilityTcIoMover := THIS^.ipTcIoMover;
END_GET
END_PROPERTY

{attribute 'monitoring':='call'}
(* Provides the current planar mover act XYZABC [mm/s] *)
PROPERTY VelocityAct : REFERENCE TO MoverVector
GET
VAR_INST
	{attribute 'hide'}
	copyOfData :  MoverVector;
END_VAR
//Creat an copy of the struct to view value in targetdbrowser and plc online view
copyOfData := THIS^.fbMover.MCTOPLC.ACT.ActVelo;
VelocityAct REF= copyOfData;
END_GET
END_PROPERTY

{attribute 'monitoring':='call'}
(* Provides the current planar mover setpoint XYZABC [mm/s] *)
PROPERTY VelocitySet : REFERENCE TO MoverVector
GET
VAR_INST
	{attribute 'hide'}
	copyOfData :  MoverVector;
END_VAR
//Creat an copy of the struct to view value in targetdbrowser and plc online view
copyOfData := THIS^.fbMover.MCTOPLC.SET.SetVelo;
VelocitySet REF= copyOfData;
END_GET
END_PROPERTY

END_FUNCTION_BLOCK

// ---- COMPONENTs/Optional/Casting/ToXpTrack.TcPOU
FUNCTION ToXpTrack : BOOL
VAR_INPUT
	iChObject : I_CH_OBJECT;
	iXpTrack : REFERENCE TO I_XP_Track;
END_VAR

VAR
	iTmp : I_XP_Track;
END_VAR

(* 
   1. Test if the interface exists
   2. Test if the object implements a "Object" interface 
   3. Write reference to interface in parameter
   4. Returne TRUE if succesfull
*)
IF iChObject <> 0 AND_THEN __QUERYINTERFACE(iChObject,iTmp) THEN
	iXpTrack := iTmp;
	ToXpTrack := TRUE;
END_IF

END_FUNCTION

// ---- FUNCTIONs/F_DistXYVectors.TcPOU
FUNCTION F_DistXYVectors : LREAL
VAR_INPUT
	pos1 : REFERENCE TO MoverVector;
	pos2 : REFERENCE TO MoverVector;
END_VAR
VAR
	fbPos2D : PositionXY;
END_VAR

IF NOT __ISVALIDREF(pos1) OR NOT __ISVALIDREF(pos2) THEN
	//Error
	F_DistXYVectors := 0;
	RETURN;
END_IF

fbPos2D.x := pos1.x - pos2.x;
fbPos2D.y := pos1.y - pos2.y;

F_DistXYVectors := fbPos2D.GetRadius();

END_FUNCTION

// ---- FUNCTIONs/F_Vector_Subtraction.TcPOU
FUNCTION F_Vector_Subtraction : MoverVector //difference.x = minuend.x - subtrahend.x
VAR_INPUT
	minuend : REFERENCE TO MoverVector;
	subtrahend : REFERENCE TO MoverVector;
END_VAR
VAR
	
END_VAR

IF NOT __ISVALIDREF(minuend) OR NOT __ISVALIDREF(subtrahend) THEN
	//Error
	RETURN;
END_IF

F_Vector_Subtraction.x	:= minuend.x	- subtrahend.x;
F_Vector_Subtraction.y	:= minuend.y	- subtrahend.y;
F_Vector_Subtraction.z	:= minuend.z	- subtrahend.z;
F_Vector_Subtraction.a	:= minuend.a	- subtrahend.a;
F_Vector_Subtraction.b	:= minuend.b	- subtrahend.b;
F_Vector_Subtraction.c	:= minuend.c	- subtrahend.c;

END_FUNCTION

// ---- FUNCTIONs/F_Vector_Multiplication.TcPOU
FUNCTION F_Vector_Multiplication : MoverVector //product.x = factor1.x * factor2.x
VAR_INPUT
	factor1 : REFERENCE TO MoverVector;
	factor2 : REFERENCE TO MoverVector;
END_VAR
VAR
	
END_VAR

IF NOT __ISVALIDREF(factor1) OR NOT __ISVALIDREF(factor2) THEN
	//Error
	RETURN;
END_IF

F_Vector_Multiplication.x	:= factor1.x	* factor2.x;
F_Vector_Multiplication.y	:= factor1.y	* factor2.y;
F_Vector_Multiplication.z	:= factor1.z	* factor2.z;
F_Vector_Multiplication.a	:= factor1.a	* factor2.a;
F_Vector_Multiplication.b	:= factor1.b	* factor2.b;
F_Vector_Multiplication.c	:= factor1.c	* factor2.c;

END_FUNCTION

// ---- FUNCTIONs/F_Vector_Addition.TcPOU
FUNCTION F_Vector_Addition : MoverVector //sum = summand1 + summand2
VAR_INPUT
	summand1 : REFERENCE TO MoverVector;
	summand2 : REFERENCE TO MoverVector;
END_VAR
VAR
	
END_VAR

IF NOT __ISVALIDREF(summand1) OR NOT __ISVALIDREF(summand2) THEN
	//Error
	RETURN;
END_IF

F_Vector_Addition.x	:= summand1.x	+ summand2.x;
F_Vector_Addition.y	:= summand1.y	+ summand2.y;
F_Vector_Addition.z	:= summand1.z	+ summand2.z;
F_Vector_Addition.a	:= summand1.a	+ summand2.a;
F_Vector_Addition.b	:= summand1.b	+ summand2.b;
F_Vector_Addition.c	:= summand1.c	+ summand2.c;

END_FUNCTION

// ---- COMPONENTs/Mover/ProductData/FB_XP_ProductData.TcPOU
FUNCTION_BLOCK FB_XP_ProductData EXTENDS FB_CH_Object IMPLEMENTS I_XP_ProductData
VAR
	{attribute 'hide'}
	ipMover : I_XP_Mover_PLC;
END_VAR

{attribute 'monitoring':='call'}
PROPERTY LinkedMover : I_XP_Mover_PLC
GET
LinkedMover := ipMover;
END_GET
END_PROPERTY

METHOD LinkToMover : BOOL //it is not necessary to call this method. This is already done internally
VAR_INPUT
	ipMoverPlc : I_XP_Mover_PLC;
END_VAR
THIS^.ipMover := ipMoverPlc;
END_METHOD

END_FUNCTION_BLOCK

// ---- COMPONENTs/Optional/Casting/ToXpMover.TcPOU
FUNCTION ToXpMover : BOOL
VAR_INPUT
	iChObject : I_CH_OBJECT;
	iXpMover : Reference to I_XP_Mover;
END_VAR

VAR
	iTmp : I_XP_Mover;
END_VAR

(* 
   1. Test if the interface exists
   2. Test if the object implements a "Object" interface 
   3. Write reference to interface in parameter
   4. Returne TRUE if succesfull
*)
IF iChObject <> 0 AND_THEN __QUERYINTERFACE(iChObject,iTmp) THEN
	iXpMover := iTmp;
	ToXpMover := TRUE;
END_IF

END_FUNCTION

// ---- COMPONENTs/Optional/Trigger/FB_XP_Trigger.TcPOU
{attribute 'no_explicit_call' := 'Do not call the body - Stick to OOP'}
FUNCTION_BLOCK FB_XP_Trigger EXTENDS FB_CH_Object IMPLEMENTS I_XP_Trigger
VAR
	{attribute 'hide'}
	bInitDone : BOOL;
	{attribute 'hide'}
	ipXpSystem : I_XP_System_Registration;
	{attribute 'hide'}
	ipAccocietedTrack : I_XP_Track;
	{attribute 'hide'}
	ipListOfMoversToCheck : CHALET_BaseComponents.I_CH_LIST;
	{attribute 'hide'}
	fTriggerPositionOnTrack : LREAL;
	{attribute 'hide'}
	eTriggerDirection : Tc3_Mc3Definitions.MC_Direction := Tc3_Mc3Definitions.MC_DIRECTION.mcDirectionPositive;
	{attribute 'hide'}
	ipMoverAtTrigger : I_XP_Mover;
	{attribute 'hide'}
	aMoversPositionLastCycle : ARRAY [0..(CHALET_BaseComponents.BaseParameterlist.MAX_OBJECTS-1)] OF LREAL; // This list is generated at the end of the PRG and contais the positions. The positions are checked in the next cycle
	{attribute 'hide'}
	aMoversTrackLastCycle : ARRAY [0..(CHALET_BaseComponents.BaseParameterlist.MAX_OBJECTS-1)] OF I_XP_Track; // This list is generated at the end of the PRG and contais the track. The tracks are checked in the next cycle
	{attribute 'hide'}
	aMoversInterfaceLastCycle : ARRAY [0..(CHALET_BaseComponents.BaseParameterlist.MAX_OBJECTS-1)] OF I_XP_Mover; // This list is generated at the end of the PRG and contais the Mover interface. The positions are checked in the next cycle
END_VAR

{attribute 'monitoring':='call'}
PROPERTY AccocietedTrack : I_XP_Track
GET
AccocietedTrack := THIS^.ipAccocietedTrack;
END_GET
SET
THIS^.ipAccocietedTrack := AccocietedTrack;
END_SET
END_PROPERTY

METHOD FB_init : BOOL
VAR_INPUT
	bInitRetains : BOOL; // if TRUE, the retain variables are initialized (warm start / cold start)
	bInCopyCode : BOOL;  // if TRUE, the instance afterwards gets moved into the copy code (online change)
	
	ipXpSystem : I_XP_System_Registration; //Interface to XTS system object
	
END_VAR
VAR_INST
	{attribute 'hide'}
	bFBInitCalledOnce : BOOL; //Do the following code once during start up and not during onlinechange
END_VAR
//Do the following code once during start up and not during onlinechange
IF NOT bFBInitCalledOnce THEN 
	;
END_IF

//Regristrate object in System if unknown
IF ipXpSystem <> 0 AND THIS^.ipXpSystem = 0 THEN
	ipXpSystem.RegisterTrigger(THIS^);
	THIS^.ipXpSystem := ipXpSystem;
END_IF

bFBInitCalledOnce := TRUE;
END_METHOD

{attribute 'monitoring':='call'}
PROPERTY HR : HRESULT
GET
IF ipAccocietedTrack <> 0 AND_THEN ipAccocietedTrack.Length > 0 THEN
	HR := S_OK;
ELSE
	HR := E_FAIL;
END_IF
END_GET
END_PROPERTY

METHOD Initialize : HRESULT
IF THIS^.ipXpSystem = 0 THEN
	//No valide interface
	Initialize := E_FAIL;
	RETURN;
END_IF


THIS^.bInitDone := TRUE;
END_METHOD

PROPERTY ListOfMoversToCheck : I_CH_List
SET
IF ListOfMoversToCheck <> 0 THEN
	ipListOfMoversToCheck := ListOfMoversToCheck;
END_IF
END_SET
END_PROPERTY

{attribute 'monitoring':='call'}
PROPERTY MoverAtTrigger : I_XP_Mover
GET
THIS^.Prepare();//Prepare Time-critical information

MoverAtTrigger := ipMoverAtTrigger;
END_GET
END_PROPERTY

{attribute 'monitoring':='call'}
PROPERTY MoverDetected : BOOL
GET
THIS^.Prepare();//Prepare Time-critical information

MoverDetected := (ipMoverAtTrigger <> 0);
END_GET
END_PROPERTY

{attribute 'monitoring':='call'}
PROPERTY PositionOnTrack : LREAL
GET
PositionOnTrack := fTriggerPositionOnTrack;
END_GET
SET
fTriggerPositionOnTrack := PositionOnTrack;
END_SET
END_PROPERTY

(* Time-critical information is processed here, which can then be polled via the property every cycle. 
The update method is usually at the end of the program and then it is already 'outdated'. *)
METHOD PRIVATE Prepare : HRESULT
VAR
	fTrackLentgh : LREAL;
	fMoverActPos,fMoverLastPos : LREAL;
	ipMoverActTrack, ipMoverLastTrack : I_XP_Track;
	fRangePositive, fRangeNegative : LREAL;
	bTriggerIsCloseAtStartTrack, bTriggerIsCloseAtEndTrack : BOOL;
	bMoverWasInRangeNeg, bMoverWasInRangePos, bMoverIsInRangeNeg, bMoverIsInRangePos : BOOL;
	bMoverIsOnSameTrack, bMoverIsOnTrackAhead, bMoverIsOnTrackBehind, bMoverWasOnTrackAhead, bMoverWasOnTrackBehind : BOOL;
	nIdx, nIdxTrack : UDINT;
	fMaxMoveDistPerCycle : LREAL; //[mm] (2 m/s(max. xPlanar speed) * 20ms(max realistic SPS cycle time) + 10%)
END_VAR
VAR_INST
	{attribute 'hide'}
	nLastUpdatedCycleCount : UDINT;
END_VAR
VAR CONSTANT
END_VAR
IF NOT bInitDone OR (THIS^.ipListOfMoversToCheck = 0) OR (THIS^.ipAccocietedTrack = 0) THEN
	Prepare := E_FAIL;
	RETURN;
END_IF

//Check if this Cycle the dates are allready prepared
IF nLastUpdatedCycleCount <> TwinCAT_SystemInfoVarList._TaskInfo[THIS^.nTaskIndex].CycleCount THEN
	nLastUpdatedCycleCount := TwinCAT_SystemInfoVarList._TaskInfo[THIS^.nTaskIndex].CycleCount;
	
	//Abort on invalide interface - Get Track length
	IF ipAccocietedTrack = 0 THEN
		RETURN;
	END_IF
	fTrackLentgh := ipAccocietedTrack.Length;
	
	//Maximum distance a mover can travel in 1 plc cycle. Worstcase 2 m/s(max. xPlanar speed) * 20ms(max realistic SPS cycle time) + 10%
	fMaxMoveDistPerCycle := 2000.0(*2000mm/s=2mm/ms*) * (TwinCAT_SystemInfoVarList._TaskInfo[THIS^.nTaskIndex].CycleTime(*[100ns]*)/10_000)(*CycleTime ms*) / 1000.0 * 1.1(*10%*);
	
	//Clear last stored Mover if an new cycle has started
	THIS^.ipMoverAtTrigger := 0;
	
	//Check old list of Moverspositions and compare them to the current position of the same mover.
	//Set Trigger if the Mover pass the Station
	fRangePositive := MIN((THIS^.fTriggerPositionOnTrack + fMaxMoveDistPerCycle),fTrackLentgh);
	fRangeNegative := MAX((THIS^.fTriggerPositionOnTrack - fMaxMoveDistPerCycle),0); 
	bTriggerIsCloseAtStartTrack := (THIS^.fTriggerPositionOnTrack - fMaxMoveDistPerCycle) < 0.0;
	bTriggerIsCloseAtEndTrack 	:= (THIS^.fTriggerPositionOnTrack + fMaxMoveDistPerCycle) > fTrackLentgh;

		
	FOR nIdx := 0 TO (CHALET_BaseComponents.BaseParameterlist.MAX_OBJECTS-1) DO
		
		IF aMoversInterfaceLastCycle[nIdx] <> 0 THEN
			fMoverActPos 			:= aMoversInterfaceLastCycle[nIdx].PositionOnTrack;
			fMoverLastPos			:= aMoversPositionLastCycle[nIdx];
			ipMoverActTrack 		:= aMoversInterfaceLastCycle[nIdx].CurrentTrack;
			ipMoverLastTrack 		:= aMoversTrackLastCycle[nIdx];
			bMoverIsOnSameTrack 	:= (ipMoverActTrack = ipAccocietedTrack);
			
			//Abort if Lasttrack is not known. Example: first cycle after enabling
			IF ipMoverActTrack = 0 OR ipMoverLastTrack = 0 THEN
				RETURN;
			END_IF
			
			//Reset flags 
			bMoverIsOnTrackAhead 	:= FALSE;		bMoverIsOnTrackBehind 	:= FALSE;		bMoverWasOnTrackAhead 	:= FALSE;		bMoverWasOnTrackBehind 	:= FALSE;
			
			//Test all tracks before and after this track to recognize that the mover has just changed tracks. 
			//This is important if this trigger is near the end or beginning of a track
			FOR nIdxTrack := 0 TO (XPlanarParameterlist.N_MAX_STATIONS_AHEAD_OR_BEHIND-1) DO
				//Tracks Ahead - Mover Is/Was on Track ahead and close(cMaxMoveDistPerCycle) at beginn on track
				IF ipMoverActTrack.TracksStartFromThis[nIdxTrack] <> 0 THEN
					bMoverIsOnTrackAhead 	:= bMoverIsOnTrackAhead 	OR ((ipAccocietedTrack = ipMoverActTrack.TracksStartFromThis[nIdxTrack])  AND ((fMoverActPos - fMaxMoveDistPerCycle) < 0.0));
					bMoverWasOnTrackAhead 	:= bMoverWasOnTrackAhead 	OR ((ipAccocietedTrack = ipMoverLastTrack.TracksStartFromThis[nIdxTrack]) AND ((fMoverLastPos - fMaxMoveDistPerCycle) < 0.0));
				END_IF
				//Tracks Behind - Mover Is/Was on Track behind and close(cMaxMoveDistPerCycle) at end on track
				IF ipMoverActTrack.TracksEndAtThis[nIdxTrack] <> 0 THEN
					bMoverIsOnTrackBehind 	:= bMoverIsOnTrackBehind 	OR ((ipAccocietedTrack = ipMoverActTrack.TracksEndAtThis[nIdxTrack])  AND ((fMoverActPos	+ fMaxMoveDistPerCycle) > ipMoverActTrack.Length));
					bMoverWasOnTrackBehind 	:= bMoverWasOnTrackBehind 	OR ((ipAccocietedTrack = ipMoverLastTrack.TracksEndAtThis[nIdxTrack]) AND ((fMoverLastPos 	+ fMaxMoveDistPerCycle) > ipMoverLastTrack.Length));
				END_IF
			END_FOR
			
			//Closed track and station in close to Modulo pos
			IF bMoverIsOnSameTrack THEN
				bMoverIsOnTrackAhead 	:= ((fMoverActPos - fMaxMoveDistPerCycle) < 0.0);
				bMoverWasOnTrackAhead 	:= ((fMoverLastPos - fMaxMoveDistPerCycle) < 0.0);
				bMoverIsOnTrackBehind 	:= ((fMoverActPos	+ fMaxMoveDistPerCycle) > ipMoverActTrack.Length);
				bMoverWasOnTrackBehind 	:= ((fMoverLastPos 	+ fMaxMoveDistPerCycle) > ipMoverLastTrack.Length);
			END_IF
			
			//Check if Mover passes the station. Ex.: If the Trigger is at Pos 0mm on track, the Mover is never in bRangeNeg. For this case check for bMoverOnTrackBefore
			bMoverIsInRangePos 		:= ((fMoverActPos >= THIS^.fTriggerPositionOnTrack) AND (fMoverActPos <= fRangePositive) AND bMoverIsOnSameTrack) OR (bMoverIsOnTrackAhead 	 AND bTriggerIsCloseAtEndTrack);   
			bMoverIsInRangeNeg 		:= ((fMoverActPos <= THIS^.fTriggerPositionOnTrack) AND (fMoverActPos >= fRangeNegative) AND bMoverIsOnSameTrack) OR (bMoverIsOnTrackBehind  AND bTriggerIsCloseAtStartTrack);     
			bMoverWasInRangePos		:= ((fMoverLastPos > THIS^.fTriggerPositionOnTrack) AND (fMoverLastPos >= fRangeNegative) AND bMoverIsOnSameTrack) OR (bMoverWasOnTrackAhead  AND bTriggerIsCloseAtEndTrack);   
			bMoverWasInRangeNeg		:= ((fMoverLastPos < THIS^.fTriggerPositionOnTrack) AND (fMoverLastPos <= fRangePositive) AND bMoverIsOnSameTrack) OR (bMoverWasOnTrackBehind AND bTriggerIsCloseAtStartTrack);     			

			IF eTriggerDirection = Tc3_Mc3Definitions.MC_DIRECTION.mcDirectionPositive  AND bMoverWasInRangeNeg AND bMoverIsInRangePos AND NOT bMoverWasInRangePos THEN
				THIS^.ipMoverAtTrigger := aMoversInterfaceLastCycle[nIdx];
				RETURN;
			ELSIF eTriggerDirection = Tc3_Mc3Definitions.MC_DIRECTION.mcDirectionNegative AND bMoverIsInRangeNeg AND bMoverWasInRangePos AND NOT bMoverWasInRangeNeg THEN
				THIS^.ipMoverAtTrigger := aMoversInterfaceLastCycle[nIdx];
				RETURN;	
			END_IF
			
		END_IF
	END_FOR
END_IF
END_METHOD

{attribute 'monitoring':='call'}
PROPERTY TimeStamp : Tc2_EtherCAT.T_DCTIME64
GET
THIS^.Prepare();//Prepare Time-critical information

///zzz todo add exact time stamp calculatioin
 IF ipMoverAtTrigger <> 0 THEN
	 TimeStamp := F_GetCurDcTaskTime64();
 ELSE
	 TimeStamp := 0;
 END_IF
END_GET
END_PROPERTY

{attribute 'monitoring':='call'}
PROPERTY TriggerDirection : Tc3_Mc3Definitions.MC_Direction
GET
TriggerDirection := eTriggerDirection;
END_GET
SET
IF TriggerDirection =Tc3_Mc3Definitions.MC_DIRECTION.mcDirectionPositive OR TriggerDirection = Tc3_Mc3Definitions.MC_DIRECTION.mcDirectionNegative THEN
	eTriggerDirection := TriggerDirection;
END_IF
END_SET
END_PROPERTY

METHOD Update : HRESULT
VAR
	nIndex : UINT;
	ipMover : I_XP_Mover;
END_VAR
//Force to do an init befor call update
IF NOT bInitDone THEN
	THIS^.Initialize();
	RETURN;
END_IF

//Clear array
MEMSET(destAddr:=ADR(aMoversInterfaceLastCycle),n:=SIZEOF(aMoversInterfaceLastCycle),fillByte:=0);
MEMSET(destAddr:=ADR(aMoversPositionLastCycle),n:=SIZEOF(aMoversPositionLastCycle),fillByte:=0);
MEMSET(destAddr:=ADR(aMoversTrackLastCycle),n:=SIZEOF(aMoversTrackLastCycle),fillByte:=0);

nIndex := 0;
IF ipListOfMoversToCheck <> 0 THEN
	THIS^.ipListOfMoversToCheck.ResetIterator();
	WHILE THIS^.ipListOfMoversToCheck.HasNextObject() DO
		
		//Cheack all Movers fill the actposition in the array
		IF ToXpMover(THIS^.ipListOfMoversToCheck.GetNextObject(),ipMover) THEN
			aMoversInterfaceLastCycle[nIndex] 	:= ipMover;
			aMoversPositionLastCycle[nIndex] 	:= ipMover.PositionOnTrack;
			aMoversTrackLastCycle[nIndex]		:= ipMover.CurrentTrack;
			nIndex := nIndex +1;
		END_IF
		
	END_WHILE	
	THIS^.ipListOfMoversToCheck.RestoreIterator();
END_IF
END_METHOD

END_FUNCTION_BLOCK

// ---- COMPONENTs/Optional/Zone/FB_XP_SoretedListOfMover.TcPOU
{attribute 'no_explicit_call' := 'Do not call the body - Stick to OOP'}
// Check zone start to end in positive direktion.
FUNCTION_BLOCK FB_XP_SoretedListOfMover EXTENDS FB_CH_Object IMPLEMENTS I_XP_Zone
VAR
	{attribute 'hide'}
	bInitDone : BOOL;
	{attribute 'hide'}
	ipXpStation : I_XP_Station; //Interface to XPlanar station 
	{attribute 'hide'}
	ipListOfMoversToCheck : CHALET_BaseComponents.I_CH_LIST;
	{attribute 'hide'}
	aMoversInZone : ARRAY [0..(CHALET_BaseComponents.BaseParameterlist.MAX_OBJECTS-1)] OF I_XP_Mover_PLC;
END_VAR

{attribute 'monitoring':='call'}
PROPERTY CtsMoversInZone : UINT
GET
VAR
	nIndex : UDINT;
END_VAR
THIS^.Prepare();//Prepare Time-critical information

//Check array for entrys, exit if fisrt empty arrayindex is found.
FOR nIndex := 0 TO (CHALET_BaseComponents.BaseParameterlist.MAX_OBJECTS-1) DO
	IF (aMoversInZone[nIndex] <> 0) THEN
		CtsMoversInZone := CtsMoversInZone +1;
	ELSE
		RETURN;
	END_IF
END_FOR
END_GET
END_PROPERTY

METHOD FB_init : BOOL
VAR_INPUT
	bInitRetains : BOOL; // if TRUE, the retain variables are initialized (warm start / cold start)
	bInCopyCode : BOOL;  // if TRUE, the instance afterwards gets moved into the copy code (online change)
	
	ipXpStation : I_XP_Station; //Interface to XPlanar station 
	ipListOfMoversToCheck : CHALET_BaseComponents.I_CH_LIST;
END_VAR
VAR_INST
	{attribute 'hide'}
	bFBInitCalledOnce : BOOL; //Do the following code once during start up and not during onlinechange
END_VAR
//Do the following code once during start up and not during onlinechange
IF NOT bFBInitCalledOnce THEN 
	;
END_IF

THIS^.ipXpStation := ipXpStation;
THIS^.ipListOfMoversToCheck := ipListOfMoversToCheck;


bFBInitCalledOnce := TRUE;
END_METHOD

METHOD Initialize : HRESULT
IF THIS^.ipXpStation = 0 THEN
	//No valide interface
	Initialize := E_FAIL;
	RETURN;
END_IF

IF THIS^.ipListOfMoversToCheck = 0 THEN
	//No valide interface
	Initialize := E_FAIL;
	RETURN;
END_IF


bInitDone := TRUE;
Initialize := S_OK;
END_METHOD

{attribute 'monitoring':='call'}
// Return a sorted list of movers in this zone. Index 0 is the mover in Front.
PROPERTY MoversInZone : REFERENCE TO ARRAY [0..(CHALET_BaseComponents.BaseParameterlist.MAX_OBJECTS-1)] OF I_XP_Mover_PLC
GET
THIS^.Prepare();//Prepare Time-critical information

MoversInZone REF= THIS^.aMoversInZone;
END_GET
END_PROPERTY

(* Time-critical information is processed here, which can then be polled via the property every cycle. 
The update method is usually at the end of the program and then it is already 'outdated'. *)
METHOD PRIVATE Prepare : HRESULT
VAR
	nLoopIndex : UDINT;
	ipMoverPlc : I_XP_Mover_PLC;
	ipMover : I_XP_Mover;
	ipPath : I_XP_Path;
	fDistToStart : LREAL;
	aDisanceToStart : ARRAY [0..(CHALET_BaseComponents.BaseParameterlist.MAX_OBJECTS-1)] OF LREAL;
END_VAR
VAR_INST
	{attribute 'hide'}
	nLastUpdatedCycleCount : UDINT;
END_VAR
IF NOT bInitDone OR ipXpStation.AccocietedTrack = 0 THEN
	Prepare := E_FAIL;
	RETURN;
END_IF

//Check if this Cycle the dates are allready prepared
IF nLastUpdatedCycleCount <> TwinCAT_SystemInfoVarList._TaskInfo[THIS^.nTaskIndex].CycleCount THEN
	nLastUpdatedCycleCount := TwinCAT_SystemInfoVarList._TaskInfo[THIS^.nTaskIndex].CycleCount;

	//Clear array
	MEMSET(destAddr:=ADR(aMoversInZone),n:=SIZEOF(aMoversInZone),fillByte:=0);
	
	//Cheack all Movers and generate a sorted list of all mover in this zone.
	THIS^.ipListOfMoversToCheck.ResetIterator();
	WHILE THIS^.ipListOfMoversToCheck.HasNextObject() DO
		//Check each mover in this stations list
		IF __QUERYINTERFACE(THIS^.ipListOfMoversToCheck.GetNextObject(),ipMoverPlc) THEN
			
			//mover and distance are known from this point and are now sorted into the array
			fDistToStart := ipMoverPlc.DistToParentStation;
			ipMoverPlc := ipMoverPlc;
			
			//Check array of movers and decide if the current one is closer to 
			FOR nLoopIndex := 0 TO (CHALET_BaseComponents.BaseParameterlist.MAX_OBJECTS-1) DO
				//empty array position
				IF aMoversInZone[nLoopIndex] = 0 THEN
					aMoversInZone[nLoopIndex] := ipMoverPlc;
					aDisanceToStart[nLoopIndex] := fDistToStart;
					EXIT;
					
				//Closer Mover found, move whole array 	
				ELSIF aDisanceToStart[nLoopIndex] > fDistToStart THEN
					MEMMOVE(srcAddr := ADR(aMoversInZone[nLoopIndex]), destAddr := ADR(aMoversInZone[nLoopIndex+1]), n := (SIZEOF(aMoversInZone[0])*(CHALET_BaseComponents.BaseParameterlist.MAX_OBJECTS-1-nLoopIndex)));
					MEMMOVE(srcAddr := ADR(aDisanceToStart[nLoopIndex]), destAddr := ADR(aDisanceToStart[nLoopIndex+1]), n := (SIZEOF(aDisanceToStart[0])*(CHALET_BaseComponents.BaseParameterlist.MAX_OBJECTS-1-nLoopIndex)));
					aMoversInZone[nLoopIndex] := ipMoverPlc;
					aDisanceToStart[nLoopIndex] := fDistToStart;
					EXIT;
					
				//check next position	
				ELSE 
					;
				END_IF
			END_FOR
		END_IF
	END_WHILE
	THIS^.ipListOfMoversToCheck.RestoreIterator();
END_IF
END_METHOD

METHOD Update : HRESULT
VAR

END_VAR
// Nothing.Check Prepare()
END_METHOD

END_FUNCTION_BLOCK

// ---- COMPONENTs/Path/FB_XP_Path.TcPOU
{attribute 'enable_dynamic_creation'}
{attribute 'no_explicit_call' := 'Do not call the body - Stick to OOP'}
FUNCTION_BLOCK FB_XP_Path EXTENDS FB_CH_Object IMPLEMENTS I_XP_Path
VAR
	fbTracksUsed : FB_CH_List;
	ipStartStation, ipDestinationStation : I_XP_Station;
	fPathLength : LREAL;
END_VAR

METHOD DistanceToDestiantion : LREAL
VAR_INPUT
	ipTrack : I_XP_Track;
	fPosOnTrack : LREAL;
END_VAR
VAR
	bCorrectPos, bCorrectTrack : BOOL;
	bPosFound : BOOL;
	fDistReturnNotOnThisTrack : LREAL;
	fStart, fEnd : LREAL;
	ipEachTrack : I_XP_Track; 
END_VAR
VAR
	//Todo add tolerance to Size >1
	fToleranceWindow : LREAL := 0.001;//[mm] if Mover is this distance mor far away from the parent, return 0mm
END_VAR
IF ipTrack = 0 THEN
	//Error -  invalide interface
	DistanceToDestiantion := CHALET_BaseComponents.GVL_Datatypes.cMaxLreal;
	RETURN;
END_IF

fDistReturnNotOnThisTrack := CHALET_BaseComponents.GVL_Datatypes.cMaxLreal;

IF (fbTracksUsed.OIDInList(ipTrack.OID) = 0) OR fPosOnTrack < 0 OR  fPosOnTrack > ipTrack.Length THEN
	//Error -  position not on track
	DistanceToDestiantion := fDistReturnNotOnThisTrack;
	RETURN;
END_IF


IF fbTracksUsed.Size = 1 THEN
	bCorrectPos := F_InLimitTest(fMinimum :=  THIS^.StationStart.PositionOnTrack, fInput:=fPosOnTrack , fMaximum:=  (THIS^.StationDestination.PositionOnTrack + fToleranceWindow));
	bCorrectTrack := (ipTrack = StationDestination.AccocietedTrack);

	IF bCorrectPos AND bCorrectTrack THEN
		DistanceToDestiantion := F_GetDistToPosModulo(fTargetPosition := THIS^.StationDestination.PositionOnTrack, fActualPosition := fPosOnTrack, fModulo := ipTrack.Length);
		//check tolerance window
		IF (DistanceToDestiantion + fToleranceWindow) >= ipTrack.Length THEN
			DistanceToDestiantion := 0.0;
		END_IF
	ELSE
		DistanceToDestiantion := fDistReturnNotOnThisTrack;
	END_IF
	RETURN;
END_IF


IF fbTracksUsed.Size > 1 THEN 
	fbTracksUsed.ResetIterator();	
	
	////First track in list
	IF ToXpTrack(fbTracksUsed.GetNextObject(),ipEachTrack) THEN
		fStart 	:= THIS^.StationStart.PositionOnTrack;
		fEnd 	:= ipEachTrack.Length;
		
		bCorrectPos := F_InLimitTest(fMinimum :=  fStart, fInput:=fPosOnTrack , fMaximum:=  fEnd);
		bCorrectTrack := (ipTrack = ipEachTrack);
		IF bCorrectPos AND bCorrectTrack THEN
			bPosFound := TRUE;
			DistanceToDestiantion := fEnd - fPosOnTrack;
		END_IF
	END_IF
	
	
	//All tracks in between
	WHILE fbTracksUsed.HasNextObject() DO
		IF ToXpTrack(fbTracksUsed.GetNextObject(),ipEachTrack) AND_THEN fbTracksUsed.HasNextObject() THEN
			fStart 	:= 0;
			fEnd 	:= ipEachTrack.Length;
			
			// still locking for the startpoint to measure the distance to Destination
			IF NOT bPosFound THEN
				bCorrectPos := F_InLimitTest(fMinimum :=  fStart, fInput:=fPosOnTrack , fMaximum:=  fEnd);
				bCorrectTrack := (ipTrack = ipEachTrack);
				IF bCorrectPos AND bCorrectTrack THEN
					bPosFound := TRUE;
					DistanceToDestiantion := fEnd - fPosOnTrack;
				END_IF
			ELSE
				// add all the tracklengths
				DistanceToDestiantion := DistanceToDestiantion + fEnd;		
			END_IF
		END_IF
	END_WHILE	
	
	
	//Last track
		fStart 	:= 0;
		fEnd 	:= (THIS^.StationDestination.PositionOnTrack + fToleranceWindow);
		// still locking for the startpoint to measure the distance to Destination
		IF NOT bPosFound THEN
			bCorrectPos := F_InLimitTest(fMinimum :=  fStart, fInput:=fPosOnTrack , fMaximum :=  fEnd);
			bCorrectTrack := (ipTrack = ipEachTrack);
			IF bCorrectPos AND bCorrectTrack THEN
				bPosFound := TRUE;
				DistanceToDestiantion := MAX(0, THIS^.StationDestination.PositionOnTrack - fPosOnTrack);
			END_IF
		ELSE
			// add all the tracklengths
			DistanceToDestiantion := DistanceToDestiantion + fEnd;		
		END_IF

	
	fbTracksUsed.RestoreIterator();
	
	IF NOT bPosFound THEN
		DistanceToDestiantion := fDistReturnNotOnThisTrack;
		RETURN;
	END_IF
END_IF
END_METHOD

{attribute 'monitoring':='call'}
//[mm]
PROPERTY Length : LREAL
GET
Length := THIS^.fPathLength;
END_GET
SET
THIS^.fPathLength := Length;
END_SET
END_PROPERTY

{attribute 'monitoring':='call'}
PROPERTY LUID : STRING //Locally unique identifier
GET
VAR
	sTempName : STRING;
END_VAR
IF ipStartStation <> 0 AND ipDestinationStation <> 0 THEN
	sTempName := CONCAT(sTempName, ipStartStation.LUID);
	sTempName := CONCAT(sTempName, ' to ' );
	sTempName := CONCAT(sTempName, ipDestinationStation.LUID);
	
ELSIF ipStartStation <> 0 THEN
	sTempName := CONCAT(sTempName, ipStartStation.LUID);
	sTempName := CONCAT(sTempName, ' to ?' );

ELSIF ipDestinationStation <> 0 THEN
	sTempName := CONCAT(sTempName, '? to ' );
	sTempName := CONCAT(sTempName, ipDestinationStation.LUID);
	
ELSE 
	sTempName := ' Unknown path';
END_IF


LUID := sTempName;
END_GET
END_PROPERTY

{attribute 'monitoring':='call'}
PROPERTY StationDestination : I_XP_Station
GET
StationDestination := THIS^.ipDestinationStation;
END_GET
SET
THIS^.ipDestinationStation := StationDestination;
END_SET
END_PROPERTY

{attribute 'monitoring':='call'}
PROPERTY StationStart  : I_XP_Station
GET
StationStart := THIS^.ipStartStation;
END_GET
SET
THIS^.ipStartStation := StationStart;
END_SET
END_PROPERTY

{attribute 'monitoring':='call'}
//List of tracks
PROPERTY TracksUsed : REFERENCE TO FB_CH_List
GET
TracksUsed REF= THIS^.fbTracksUsed;
END_GET
END_PROPERTY

END_FUNCTION_BLOCK

// ---- FUNCTIONs/F_InLimitTest.TcPOU
FUNCTION F_InLimitTest : BOOL
VAR_INPUT
	fMinimum 	: LREAL;
	fMaximum 	: LREAL;
	fInput 		: LREAL;
END_VAR

//Normal case
// 9 Max
// 5 Test
// 1 Min
IF fMinimum <= fMaximum THEN
	F_InLimitTest := (fInput >= fMinimum) AND (fInput <= fMaximum);
	
//Modulo case	
// 6 | 6  Max
// 5 | 9  Test
// 8 | 8  Min
ELSIF fMinimum > fMaximum THEN
	F_InLimitTest := NOT((fInput > fMaximum) AND (fInput < fMinimum));
END_IF

END_FUNCTION

// ---- FUNCTIONs/F_GetDistToPosModulo.TcPOU
FUNCTION F_GetDistToPosModulo : LREAL //This is only working in Positiv Direktion
VAR_INPUT
	fTargetPosition : LREAL;
	fActualPosition : LREAL;
	fModulo 		: LREAL;
END_VAR

VAR

END_VAR

IF fTargetPosition < fActualPosition THEN
	fTargetPosition := fTargetPosition + fModulo;
END_IF

F_GetDistToPosModulo := fTargetPosition - fActualPosition;

END_FUNCTION

// ---- COMPONENTs/Stationen/A-Star-Node/FB_AStarNode.TcPOU
FUNCTION_BLOCK FB_AStarNode EXTENDS FB_CH_Object IMPLEMENTS I_PathAStarNode
VAR
	{attribute 'hide'}  
	ipStation : I_XP_Station;
	{attribute 'hide'}  
	fbRouteUsedToNode : FB_CH_LIST;	
END_VAR

{attribute 'monitoring':='call'}
PROPERTY LUID : STRING
GET
IF THIS^.Station <> 0 THEN
	LUID := THIS^.Station.LUID;
END_IF
END_GET
END_PROPERTY

{attribute 'monitoring':='call'}
PROPERTY PathLength : LREAL
GET
VAR
	ipEachPath : I_XP_Path;
END_VAR
PathLength := 0.0;


fbRouteUsedToNode.ResetIterator();
WHILE fbRouteUsedToNode.HasNextObject() DO
	IF __QUERYINTERFACE(fbRouteUsedToNode.GetNextObject(), ipEachPath) THEN
		PathLength := PathLength + ipEachPath.Length;
	END_IF
END_WHILE
fbRouteUsedToNode.RestoreIterator();
END_GET
END_PROPERTY

{attribute 'monitoring':='call'}
PROPERTY RouteUsedToNode : REFERENCE TO FB_CH_List
GET
RouteUsedToNode REF= fbRouteUsedToNode;
END_GET
END_PROPERTY

//here in this case the SortOrder is used to get the shortest path. 
PROPERTY SortOrderInList : UDINT
GET
SortOrderInList := TO_UDINT(THIS^.PathLength);
END_GET
END_PROPERTY

{attribute 'monitoring':='call'}
PROPERTY Station : I_XP_Station
GET
Station := ipStation;
END_GET
SET
ipStation := Station;
END_SET
END_PROPERTY

END_FUNCTION_BLOCK

// ---- COMPONENTs/Stationen/FB_XP_Station.TcPOU
{attribute 'enable_dynamic_creation'}
{attribute 'no_explicit_call' := 'Do not call the body - Stick to OOP'}
(* XPlanar station - n per associated XPlanar. Can be instantiated as an array and/or individually
	The stations are the main component of the application. As soon as the system has been started up and all movers are on the track, the movers are only sent from one station to the next.
	Parameters:
		xPos, yPos 			= Absolute position of the station on the xPlanar.
		ipAccocietedTrack 	= The track on which the station is located. If the XY position is not on this track, the next possible track position is assumed on this track.
		sUniqueName 		= Unique name that may only exist once.
		sTargetGroup 		= A name for a group to which this station belongs. Important for redundant stations
 *)	
FUNCTION_BLOCK FB_XP_Station EXTENDS FB_CH_Object IMPLEMENTS I_XP_Station, I_XP_Station_PLC
VAR
	//optional - To visualize the station position in LiveView
	fbOptionalTrackUsedInLiveView : MC_PlanarTrack;

	{attribute 'hide'}
	bErrorDuringFbInit : BOOL;	//Fatal error - Not possible to reset
	
	{attribute 'hide'}
	bInitDone : BOOL;
	{attribute 'hide'}	
	bTrackIsSetInFbInit : BOOL;
	{attribute 'hide'}	
	bMoversInPlace : BOOL;
	{attribute 'hide'}                   	
	eActiveCommand 		: CHALET_Nc.E_NcAxisCommands := CHALET_Nc.E_NcAxisCommands.None;
	{attribute 'hide'}	
	ipXpSystem : I_XP_System_Registration;
	{attribute 'hide'}
	bReadyToRecvMovers 		: BOOL := TRUE;
	{attribute 'hide'}
	nCtsMoversMustLeaveThisStation : UDINT;
	{attribute 'hide'}
	sTargetGroup 				: STRING;
	
	{attribute 'hide'}
	bSuppressDynamicsChange		: BOOL; // Suppress to change the dynamic(Gap+velocity) of passing movers. This is usefull in startup
	{attribute 'hide'}
	fMoverGapAtExit 			: LREAL := XPlanarParameterlist.F_GAP_DEFAULT; // Every mover that leaves or passes the station gets this new gap as a target.
	{attribute 'hide'}	
	fbPositionPlanned : PositionXY; //this is the configured/planned position of the station. set via FB_init. If it is not on the track, the PosOnTrackXY is different
	{attribute 'hide'}	
	fPositionOnTrack : LREAL;
	{attribute 'hide'}
	fbPositionOnTrackXY : PositionXY;	
	{attribute 'hide'}	
	nState_Configuring: INT;
	{attribute 'hide'}	
	ipAccocietedTrack : I_XP_Track;
	{attribute 'hide'}
	nMoverQueueSize 			: UINT;
	{attribute 'hide'}
	fTargetPosWindow			: LREAL := 0.05; //[mm]
	{attribute 'hide'}
	tTargetPosMonitoringTime	: TIME := T#0MS;

	
	(*List of stations*)
	{attribute 'hide'}	
	fbStationsAhead : FB_CH_List;
	{attribute 'hide'}	
	fbStationsBehinde : FB_CH_List;
	
	(*List of paths*)
	{attribute 'hide'}	
	fbListPathAhead : FB_CH_List;
	{attribute 'hide'}
	fbListPathBehind : FB_CH_List;
	
	(* Lists to handle the ownership of movers *)
	{attribute 'hide'}
	fbAssignedMovers 			: FB_CH_List;		// Movers approaching the station. This station is the parent of this movers
	{attribute 'hide'}
	fbFeedback : FB_CH_Feedback(ipSourceInfo := fbSourceInfo);		
	
	//Simulation
	{attribute 'hide'}
	fSimulationProcessDuration 	: LREAL; //[s]
	{attribute 'hide'}
	sSimulationTargetStation	: STRING; //GroupID of the target station to automatic send after the duration
	
	
	//ipXpSystem Is Not Valid at this point, call the konstruktor again in the FB_Init
	{attribute 'hide'}
	fbTrigger 					: FB_XP_Trigger(ipXpSystem);
	{attribute 'hide'}
	fbSortedListMoversInQueue	: FB_XP_SoretedListOfMover(	ipXpStation := THIS^,
															ipListOfMoversToCheck := fbAssignedMovers );
	{attribute 'hide'}
	fDecisionDistance: LREAL;//[mm]
	{attribute 'hide'}
	bNetworkHasTrackBranches : BOOL;//True if atleas on branche is existing in network
	{attribute 'hide'}
	sFilter : STRING :=  XPlanarParameterlist.S_ANY_STATION_NAME;
	{attribute 'hide'}	
	fbAlarmStationIsBlocked : FB_TcAlarm;
END_VAR

// Dynamic to use if an Mvoer passes the station
// Every mover that leaves or passes the station gets this new velo as a target.
VAR
	{attribute 'hide'}	
	fMoverVeloAtExit : MC_LREAL := MC_DEFAULT; //equivalent to data type LREAL + MC_DEFAULT, MC_MAXIMUM
	{attribute 'hide'}	
    fMoverAccAtExit : MC_LREAL := MC_DEFAULT; //equivalent to data type LREAL + MC_DEFAULT, MC_MAXIMUM
	{attribute 'hide'}	
    fMoverDecAtExit : MC_LREAL := MC_DEFAULT; //equivalent to data type LREAL + MC_DEFAULT, MC_MAXIMUM
END_VAR

{attribute 'monitoring':='call'}
//Track on which the station is located
PROPERTY AccocietedTrack : I_XP_Track
GET
AccocietedTrack := THIS^.ipAccocietedTrack;
END_GET
END_PROPERTY

METHOD AddMoverToQueue : HRESULT
VAR_INPUT
	ipMover : I_XP_Mover;
END_VAR
//Get I_CH_Objekt of mover to put it in to a list.
IF ipMover <> 0 THEN
	//Add in List of Movers in this station
	THIS^.fbAssignedMovers.AddObject(ipMover);
	
	//Handover information in Mover
	ipMover.ParentStation := (THIS^);

	AddMoverToQueue := S_OK;
ELSE
	AddMoverToQueue := E_FAIL;;	
END_IF
END_METHOD

{attribute 'monitoring':='call'}
//List of movers managed by this station
PROPERTY AssignedMovers : I_CH_List
GET
AssignedMovers := THIS^.fbAssignedMovers;
END_GET
END_PROPERTY

METHOD PROTECTED CheckInvalideParameter : HRESULT
VAR
 	ipStation : I_XP_Station;
	fbListOfStationsToCheck : FB_CH_List;
END_VAR
VAR_INST
	{attribute 'hide'}	
	fbAlarm : FB_TcAlarm;
END_VAR
//Get a list of all station whitout this station
fbListOfStationsToCheck.Duplicate(THIS^.ipXpSystem.StationsUsed);
fbListOfStationsToCheck.RemoveObject(THIS^);


fbListOfStationsToCheck.ResetIterator();
WHILE fbListOfStationsToCheck.HasNextObject() DO
	IF ToXpStation(fbListOfStationsToCheck.GetNextObject(), ipStation) THEN
		
		//Check for same positions
		IF (ipStation.PositionOnTrack = THIS^.PositionOnTrack) AND (ipStation.AccocietedTrack = THIS^.AccocietedTrack)  THEN
			//Error two stations have same position on track
			CheckInvalideParameter := E_FAIL;
			IF NOT fbAlarm.bRaised THEN
				fbAlarm.CreateEx(stEventEntry:=TC_EVENTS.CHALET_XPlanar_Events.DuplicateStationPositions, ipSourceInfo := THIS^.fbSourceInfo, bWithConfirmation := FALSE);
				fbAlarm.ipArguments.AddStringByValue(THIS^.LUID).AddStringByValue(ipStation.LUID);
				fbAlarm.Raise(0);			
			END_IF
			RETURN;
		END_IF
		
		//Check same unique id
		IF (ipStation.LUID = THIS^.LUID) THEN
			//Error two stations have same unique id
			CheckInvalideParameter := E_FAIL;
			IF NOT fbAlarm.bRaised THEN
				fbAlarm.CreateEx(stEventEntry:=TC_EVENTS.CHALET_XPlanar_Events.DuplicateStationName, ipSourceInfo := THIS^.fbSourceInfo, bWithConfirmation := FALSE);
				fbAlarm.ipArguments.AddStringByValue(THIS^.LUID);
				fbAlarm.Raise(0);			
			END_IF
			RETURN;
		END_IF
		
		fbListOfStationsToCheck.RemoveObject(ipStation);
	END_IF
END_WHILE
END_METHOD

//Call this Methode whith seq 0->99, and wait each step until S_OK is returned
METHOD Configure : HRESULT
VAR_INPUT
	nSeq : UINT; //0->100
END_VAR

VAR_INST
	{attribute 'hide'}
	fbFeedback : MC_PlanarFeedback;	
END_VAR
VAR
	bOptionalTrackUsedInLiveViewIsMapped : BOOL;
	fbPositionXYC : PositionXYC;
	ipEachTrack : I_XP_Track;
END_VAR
bOptionalTrackUsedInLiveViewIsMapped := fbOptionalTrackUsedInLiveView.MCTOPLC_STD.TrackOID <> 0;

CASE nSeq OF
	5:	//Get interface of trackobject
		Configure := THIS^.GetAccocietedTrack();	

	10: //Get closest XY-Position on track
		Configure := THIS^.GetPosOnTrack();
		
	11:	//Automatic add/remove this station from list of all station if it is createt automatic at the end of each track and is (not) used	
		Configure := THIS^.ManageAutomaticallyGeneratedStations();
		
	12: //Check id is unique and not multiple stations at same position
		Configure := THIS^.CheckInvalideParameter();		
				
	13:	//Init Tigger
		fbTrigger.AccocietedTrack := THIS^.AccocietedTrack;
		fbTrigger.PositionOnTrack := THIS^.PositionOnTrack;
		fbTrigger.ListOfMoversToCheck := THIS^.ipXpSystem.MoversPresent;//All mover
		fbTrigger.TriggerDirection := Tc3_Mc3Definitions. MC_DIRECTION.mcDirectionPositive;
		Configure := fbTrigger.Initialize();
	
	14:	//Init Zone		
		Configure := fbSortedListMoversInQueue.Initialize();	
	
	20: //Fill the list of all paths before this station
		Configure := THIS^.GetPathsAhead();		
		
	25: //Fill the list of all stations before this station
		Configure := THIS^.GetStationAhead();

	30: //Fill the list of all paths behinde this station
		Configure := THIS^.GetStationBehinde();	
			
	35: //Fill the list of all stations behinde this station
		Configure := THIS^.GetPathsBehind();

	40: //Determine the distance from which the station can give a new command to a mover
		Configure := THIS^.GetDecisionDistance();
		

//----------------------------------------------------------------		
//The station can optionally be linked to a track object. this track is then displayed in the live view.
//It takes several cycles to prepare the object
	80: IF bOptionalTrackUsedInLiveViewIsMapped THEN
			fbOptionalTrackUsedInLiveView.Clear(fbFeedback);
		END_IF
		
	81:	//Wait for clearing
		IF bOptionalTrackUsedInLiveViewIsMapped THEN
			IF fbFeedback.Done THEN
				Configure := S_OK;
			ELSIF fbFeedback.Busy THEN
				Configure := S_PENDING;
			ELSIF fbFeedback.Error THEN
				Configure := E_FAIL;
			END_IF	
		END_IF

	82: //Set position 
		IF bOptionalTrackUsedInLiveViewIsMapped THEN
			fbPositionXYC.SetValuesXY(THIS^.PositionOnTrackXY.x, THIS^.PositionOnTrackXY.y);
			fbOptionalTrackUsedInLiveView.AppendPosition(position := fbPositionXYC, commandFeedback:= fbFeedback);	
		END_IF	
	
	83:	//Wait for set position
		IF bOptionalTrackUsedInLiveViewIsMapped THEN
			IF fbFeedback.Done THEN
				Configure := S_OK;
			ELSIF fbFeedback.Busy THEN
				Configure := S_PENDING;
			ELSIF fbFeedback.Error THEN
				Configure := E_FAIL;
			END_IF	
		END_IF
		
	84:	//Set name of "track" to stationsname 
		IF bOptionalTrackUsedInLiveViewIsMapped THEN
 			Configure := SetTrackObjName();
		END_IF
//----------------------------------------------------------------

	90: //Create some internal used variable
		THIS^.bNetworkHasTrackBranches := FALSE;
		THIS^.ipXpSystem.Tracks.ResetIterator();
		WHILE THIS^.ipXpSystem.Tracks.HasNextObject() DO
			IF __QUERYINTERFACE(THIS^.ipXpSystem.Tracks.GetNextObject(), ipEachTrack) AND_THEN (ipEachTrack.TracksAhead.Size > 1) THEN
				THIS^.bNetworkHasTrackBranches := TRUE;
				EXIT;
			END_IF
		END_WHILE
		THIS^.ipXpSystem.Tracks.RestoreIterator();
		
		

	100..CHALET_BaseComponents.GVL_Datatypes.cMaxUint: 
		// 100..MaxUint -> Invalide input
		Configure := E_FAIL;
		
	ELSE 
		//If an step is not defind/used return ok
		Configure := S_OK;
END_CASE


fbOptionalTrackUsedInLiveView.Update();
fbFeedback.Update();
END_METHOD

{attribute 'monitoring':='call'}
PROPERTY CtsEmptySpaceInQueue : UDINT
GET
//Handle UINT Overflow
IF THIS^.fbAssignedMovers.Size >= THIS^.nMoverQueueSize THEN
	CtsEmptySpaceInQueue := 0;
ELSE 
	CtsEmptySpaceInQueue := THIS^.nMoverQueueSize - THIS^.fbAssignedMovers.Size;
END_IF
END_GET
END_PROPERTY

{attribute 'monitoring':='call'}
PROPERTY CtsMoversInQueue : UDINT
GET
CtsMoversInQueue := THIS^.fbAssignedMovers.Size;
END_GET
END_PROPERTY

{attribute 'monitoring':='call'}
(*[mm]
As soon as the mover is closer than this distance, the mover can be sent on to the next one if necessary.
This is the distance from the station to the end of the track or the shortest path to this station. Depending on which is closer. This is to ensure that the mover can no longer be overhauled.
This proberty can make the internal calculated distance smaller but not larger
Recalculated each disable/enable of the system*)
//Todo Increase shpuld also be possible
PROPERTY DecisionDistance : LREAL
GET
DecisionDistance := THIS^.fDecisionDistance;
END_GET
SET
THIS^.fDecisionDistance := MIN(THIS^.fDecisionDistance, ABS(DecisionDistance));
END_SET
END_PROPERTY

METHOD DeleteMoversQueue : HRESULT
VAR
	ipTempMover : I_XP_Mover;
END_VAR
//Not allowed in enabled state
IF THIS^.ipXPSystem.Enabled THEN
	DeleteMoversQueue := E_FAIL;
	RETURN;
END_IF


//Delete intormation in linked mover
THIS^.fbAssignedMovers.ResetIterator();
WHILE THIS^.fbAssignedMovers.HasNextObject() DO
	IF ToXPMover(THIS^.fbAssignedMovers.GetNextObject(),ipTempMover) THEN
		ipTempMover.ParentStation := 0;
	END_IF	
END_WHILE

//Clear list
fbAssignedMovers.Clear();

DeleteMoversQueue := S_OK;
END_METHOD

//This method is called when the system is disabled. Links are deleted as they may no longer be valid
METHOD Disassemble : HRESULT
VAR_INPUT
END_VAR
fbStationsAhead.Clear(); 
fbStationsBehinde.Clear(); 
fbListPathAhead.Clear(); 
fbListPathBehind.Clear(); 

Disassemble := S_OK;
END_METHOD

METHOD FB_exit : BOOL
VAR_INPUT
	bInCopyCode : BOOL; // if TRUE, the exit method is called for exiting an instance that is copied afterwards (online change).
END_VAR
VAR
	pFbPath : POINTER TO FB_XP_Path;
	ipObject : I_CH_Object;
END_VAR
// Not in an onlinechange - only in switch to configmode
IF NOT bInCopyCode THEN
	
	//Clear list, delete dynamic_creation path objects
	WHILE NOT THIS^.fbListPathAhead.IsEmpty DO
		ipObject := fbListPathAhead.GetRandomObject();
		fbListPathAhead.RemoveObject(ipObject);
		
		//Get pointer and delete
		IF __QUERYPOINTER(ipObject, pFbPath) THEN
			__DELETE(pFbPath);
		END_IF
	END_WHILE

END_IF
END_METHOD

METHOD FB_init : BOOL
VAR_INPUT
	bInitRetains : BOOL; // if TRUE, the retain variables are initialized (warm start / cold start)
	bInCopyCode : BOOL;  // if TRUE, the instance afterwards gets moved into the copy code (online change)
	
	ipSystem 			: I_CH_Object;
	ipAccocietedTrack 	: I_XP_Track;//track on which the station is located
	sUniqueName			: STRING;		//expl.:'Loading' unique identification for this station
	sTargetGroup		: STRING;	//to which group of stations does this station belong? e.g. several stations can belong to one 'Infeed' if this is implemented redundantly.
	nMoverQueueSize 	: UINT;
	xPos				: LREAL; 	
	yPos				: LREAL; 	
END_VAR
VAR 

END_VAR
//Do the following code once during start up and not during onlinechange
IF NOT bInCopyCode THEN 
	bErrorDuringFbInit := FALSE;
	
	(* Register to the Xplanar System
	   1. Test if the interface exists
	   2. Test if the object implements a "System for Mover" interface 
	*)
	IF ipSystem <> 0 AND_THEN __QUERYINTERFACE(ipSystem,THIS^.ipXpSystem) THEN
		THIS^.ipXpSystem.RegisterStation(THIS^);
	ELSE
		bErrorDuringFbInit := TRUE;
	END_IF

	THIS^.fbFeedback.ActiveCommand 		:= TO_STRING(THIS^.eActiveCommand);	
	
	// 0 = get closest track (in step configure)
	IF ipAccocietedTrack <> 0 THEN
		THIS^.ipAccocietedTrack := ipAccocietedTrack;
		bTrackIsSetInFbInit := TRUE;
	END_IF
	 
	
	//"" is maybe entered in an waiting or dynamic station and the name is not important
	IF sUniqueName <> '' THEN 
		THIS^.fbSourceInfo.sName := sUniqueName;
	ELSE
		sUniqueName := THIS^.fbSourceInfo.sName;
	END_IF

	
	//"" is maybe entered in an waiting or dynamic station and the name is not important
	IF sTargetGroup <> '' THEN 
		THIS^.sTargetGroup := sTargetGroup;
	ELSE
		THIS^.sTargetGroup := THIS^.fbSourceInfo.sName;
	END_IF

	
	THIS^.nMoverQueueSize 		:= nMoverQueueSize;
	THIS^.fbPositionPlanned.x 	:= xPos;
	THIS^.fbPositionPlanned.y 	:= yPos;


	THIS^.fbTrigger.FB_init(FALSE,FALSE, THIS^.ipXpSystem);

END_IF
END_METHOD

{attribute 'monitoring':='call'}
PROPERTY Feedback : I_CH_Feedback
GET
Feedback := THIS^.fbFeedback;
END_GET
END_PROPERTY

{attribute 'monitoring':='call'}
//Filter content, movers with one of these targets may not approach or drive over the station
PROPERTY Filter : STRING
GET
Filter := sFilter;
END_GET
SET
sFilter := Filter;
END_SET
END_PROPERTY

METHOD protected GetAccocietedTrack : HRESULT
VAR
	ipTrack : I_XP_Track;

	fPosOnTrack, fDist	: LREAL;
	fbPositionXYC : PositionXYC;
	fbPositionXY : PositionXY;
	ipClosestTrack : I_XP_Track;
	fDistClosestTrack : LREAL := CHALET_BaseComponents.GVL_Datatypes.cMaxLreal;
END_VAR
//If track is not defind during FB_init, get closest track 
IF NOT bTrackIsSetInFbInit THEN
	THIS^.ipAccocietedTrack := 0;
	THIS^.ipXpSystem.Tracks.ResetIterator();
	WHILE THIS^.ipXpSystem.Tracks.HasNextObject() DO
		IF ToXpTrack(THIS^.ipXpSystem.Tracks.GetNextObject(),ipTrack) THEN 
			
			fPosOnTrack := ipTrack.PlanarTrack.GetArcLengthClosestTo(geometry:= THIS^.fbPositionPlanned);
			//Get the XYC Pos on track
			ipTrack.PlanarTrack.GetPositionAt(fPosOnTrack, fbPositionXYC);
			//Get radius/ distance to positionTarget
			fbPositionXY.x  := THIS^.fbPositionPlanned.x - fbPositionXYC.x;
			fbPositionXY.y  := THIS^.fbPositionPlanned.y - fbPositionXYC.y;
			fDist := fbPositionXY.GetRadius();
			
			IF fDist < fDistClosestTrack THEN
				fDistClosestTrack := fDist;
				ipClosestTrack := ipTrack;
			END_IF
		END_IF
	END_WHILE
	THIS^.ipXpSystem.Tracks.RestoreIterator();
	
	
	THIS^.ipAccocietedTrack := ipClosestTrack;	
END_IF

// Error - No track found
IF THIS^.ipAccocietedTrack = 0 THEN
	GetAccocietedTrack := E_FAIL;
	RETURN;
END_IF
END_METHOD

METHOD GetDecisionDistance : HRESULT
VAR
	fDistToStartOfTrack : LREAL := CHALET_BaseComponents.GVL_Datatypes.cMaxLreal;
	fDistStationBehind : LREAL := CHALET_BaseComponents.GVL_Datatypes.cMaxLreal;
	
	ipPath : I_XP_Path;
END_VAR
(*
As soon as the mover is closer than this distance, the mover can be sent on to the next one if necessary.
This is the distance from the station to the end of the track or the shortest path to this station. Depending on which is closer. This is to ensure that the mover can no longer be overhauled.
*)
fDistToStartOfTrack := THIS^.PositionOnTrack;

THIS^.PathsBehinde.ResetIterator();
WHILE THIS^.PathsBehinde.HasNextObject() DO
	IF __QUERYINTERFACE(THIS^.PathsBehinde.GetNextObject(), ipPath) THEN
		fDistStationBehind := MIN(fDistStationBehind, ipPath.Length);
	END_IF
END_WHILE
THIS^.PathsBehinde.RestoreIterator();

THIS^.fDecisionDistance := CHALET_BaseComponents.GVL_Datatypes.cMaxLreal;
THIS^.fDecisionDistance := MIN(THIS^.fDecisionDistance, (fDistToStartOfTrack - 1.0));
THIS^.fDecisionDistance := MIN(THIS^.fDecisionDistance, (fDistStationBehind - 1.0));
THIS^.fDecisionDistance := MIN(THIS^.fDecisionDistance, XPlanarParameterlist.F_DIST_SET_NEW_MOVE_CMD_BEFORE_REACHING_PARENT_STATION);


IF THIS^.fDecisionDistance < 1.0 THEN 
	THIS^.fDecisionDistance := 1.0;
END_IF

GetDecisionDistance := S_OK;
END_METHOD

METHOD protected GetPathsAhead : HRESULT
VAR_INPUT
END_VAR

VAR
	fbPathElementsToCheck : FB_CH_List;
	fbListStationsToGetClosest : FB_CH_List;	
	ipObjectPathAhead 				: I_CH_Object;
	ipStation,ipStation1,ipStation2 	: I_XP_Station;
	ipTrack					: I_XP_Track; 
	ipLastAddedTrack 		: I_XP_Track;
	ipPath 					: I_XP_Path;
	ipPathCurrentLoop  		: I_XP_Path;
	
	
	pFbPath, pFbPathCurrentLoop : POINTER TO FB_XP_Path;
	
	fSeachStartPoint : LREAL;
	nIdx : UDINT;
END_VAR
(*
Check whether there is a station further ahead on this track than this one.
If there is no other station on the track, the previous tracks are filled into a list and searched one after the other to see if they have valid stations. 
If the tracks also have no stations, the track before it is added to the list,...
*)

//Clear list, delete dynamic_creation path objects
WHILE NOT fbListPathAhead.IsEmpty DO
	ipObjectPathAhead := fbListPathAhead.GetRandomObject();
	fbListPathAhead.RemoveObject(ipObjectPathAhead);
	
	//get pointer and delete
	IF __QUERYPOINTER(ipObjectPathAhead, pFbPath) THEN
		__DELETE(pFbPath);
	END_IF	
		
END_WHILE


//new dynamic_creation path objects
pFbPath := __NEW(FB_XP_Path);
//init path
pFbPath^.StationStart := THIS^;
pFbPath^.TracksUsed.ResetIterator();
pFbPath^.TracksUsed.AddObject(THIS^.AccocietedTrack);

//add to list
fbPathElementsToCheck.AddObject(pFbPath^);

//On first pathsearch get an Station who is further ahead than this
fSeachStartPoint := THIS^.PositionOnTrack;



//While list is not empty
WHILE NOT fbPathElementsToCheck.IsEmpty DO
	__QUERYINTERFACE(fbPathElementsToCheck.GetRandomObject(), ipPathCurrentLoop);
	__QUERYINTERFACE(ipPathCurrentLoop.TracksUsed.GetNextObject(),ipLastAddedTrack);
	
	
	//Closed loop
	IF ipLastAddedTrack.ClosedLoop THEN
		//on closed-loop add all stations of this track to list
		fbListStationsToGetClosest.Duplicate(ipLastAddedTrack.StationsOnTrack);
	
		//remove THIS station from list if more than on station is existing
		IF fbListStationsToGetClosest.Size > 1 THEN
			fbListStationsToGetClosest.RemoveObject(THIS^);
		END_IF
	
		
	
	ELSE
		//Not closed loop	
		//Get a List of all stations on track Position > Startpoint
		ipLastAddedTrack.StationsOnTrack.ResetIterator();
		fbListStationsToGetClosest.Clear();
		WHILE ipLastAddedTrack.StationsOnTrack.HasNextObject() DO
			IF ToXpStation(ipLastAddedTrack.StationsOnTrack.GetNextObject(),ipStation) THEN
				//Add all station ahead to list. on closed-loop add all stations of this track to list
				IF ipStation.PositionOnTrack > fSeachStartPoint THEN
					fbListStationsToGetClosest.AddObject(ipStation);
				END_IF
			END_IF
		END_WHILE	
	END_IF
		
	

	
	//Get closest to startpos(0mm)
	WHILE fbListStationsToGetClosest.Size > 1 DO
		fbListStationsToGetClosest.ResetIterator();
		__QUERYINTERFACE(fbListStationsToGetClosest.GetNextObject(),ipStation1);
		__QUERYINTERFACE(fbListStationsToGetClosest.GetNextObject(),ipStation2);
		
		//If station1 is closer to start than station2, remove station2
		IF 		F_GetDistToPosModulo(fTargetPosition := ipStation1.PositionOnTrack, fActualPosition := fSeachStartPoint, fModulo := ipLastAddedTrack.Length) 
			< 	F_GetDistToPosModulo(fTargetPosition := ipStation2.PositionOnTrack, fActualPosition := fSeachStartPoint, fModulo := ipLastAddedTrack.Length) THEN
			fbListStationsToGetClosest.RemoveObject(ipStation2);
		ELSE	
			fbListStationsToGetClosest.RemoveObject(ipStation1);
		END_IF
	END_WHILE
	
	
	IF fbListStationsToGetClosest.Size = 1 THEN
		//Station FOUND
		__QUERYINTERFACE(fbListStationsToGetClosest.GetRandomObject(), ipStation);
		ipPathCurrentLoop.StationDestination := ipStation;
		
		//Calculate Tracklentgh
		ipPathCurrentLoop.TracksUsed.ResetIterator();
		WHILE ipPathCurrentLoop.TracksUsed.HasNextObject() DO
			IF ToXpTrack(ipPathCurrentLoop.TracksUsed.GetNextObject(),ipTrack) THEN
				ipPathCurrentLoop.Length := ipPathCurrentLoop.Length + ipTrack.Length;
			END_IF
		END_WHILE	
		ipPathCurrentLoop.Length := ipPathCurrentLoop.Length - ipPathCurrentLoop.StationStart.PositionOnTrack;
		ipPathCurrentLoop.Length := ipPathCurrentLoop.Length - ipPathCurrentLoop.StationDestination.AccocietedTrack.Length + ipPathCurrentLoop.StationDestination.PositionOnTrack;
		
		//Modulo on cloosed track add 1 track length 
		IF ipPathCurrentLoop.StationStart.AccocietedTrack = ipPathCurrentLoop.StationDestination.AccocietedTrack AND 
			ipPathCurrentLoop.StationStart.PositionOnTrack > ipPathCurrentLoop.StationDestination.PositionOnTrack THEN
				ipPathCurrentLoop.Length := ipPathCurrentLoop.Length + ipPathCurrentLoop.StationDestination.AccocietedTrack.Length;
		END_IF
		
		fbListPathAhead.AddObject(ipPathCurrentLoop);
		fbPathElementsToCheck.RemoveObject(ipPathCurrentLoop);
	ELSE
		//Station NOT-FOUND, add the subsequent tracks in the list
		ipLastAddedTrack.TracksAhead.ResetIterator();
		WHILE ipLastAddedTrack.TracksAhead.HasNextObject() DO
			ToXpTrack(ipLastAddedTrack.TracksAhead.GetNextObject(), ipTrack);
			//dublicate current path
			pFbPath := __NEW(FB_XP_Path);
			//Get pointer from fb behinde this interface
			__QUERYPOINTER(ipPathCurrentLoop, pFbPathCurrentLoop);
			MEMCPY(destAddr := pFbPath, srcAddr := pFbPathCurrentLoop, n := SIZEOF(FB_XP_Path));
			//Add the new track to fresh created path
			pFbPath^.TracksUsed.AddObject(ipTrack);
			//Add to list to check
			fbPathElementsToCheck.AddObject(pFbPath^);
			
		END_WHILE

		
		//delete current path
		fbPathElementsToCheck.RemoveObject(ipPathCurrentLoop);

		//get pointer and delete
		IF __QUERYPOINTER(ipPathCurrentLoop, pFbPath) THEN
			__DELETE(pFbPath);
		END_IF	
		
	END_IF

	fSeachStartPoint := -0.1;
END_WHILE
END_METHOD

METHOD protected GetPathsBehind : HRESULT
VAR
	ipThisStation : I_XP_Station;
	ipXpStation : I_XP_Station;
	ipPath		: I_XP_Path;
END_VAR
ipThisStation := THIS^;
fbListPathBehind.Clear();

THIS^.fbStationsBehinde.ResetIterator();
WHILE THIS^.fbStationsBehinde.HasNextObject() DO
	IF __QUERYINTERFACE(THIS^.fbStationsBehinde.GetNextObject(),ipXpStation) THEN
		ipXpStation.PathsAhead.ResetIterator();
		WHILE ipXpStation.PathsAhead.HasNextObject() DO
			IF __QUERYINTERFACE(ipXpStation.PathsAhead.GetNextObject(),ipPath) AND_THEN ipPath.StationDestination = ipThisStation THEN
				//add path to this station to list
				fbListPathBehind.AddObject(ipPath);
			END_IF
		END_WHILE	
	END_IF
END_WHILE
END_METHOD

(*THIS METHOD uses the A* algorithm TO find the shortest route TO the destination in the network. Returns an INTERFACE with information about the destination found, such as station, path TO destination, path length.
If an interface=0 is returned, then no path can be found at the current time.*)
METHOD GetPathToTarget : I_PathAStarNode
VAR_INPUT
	sTargetStation : REFERENCE TO STRING; //unique station name or group of stations. EmptyString=Any
END_VAR
VAR	
	nDifZero : INT;	///zzz remove

	nIdx : UDINT;
	bCorrectLUID: BOOL;
	bCorrectGroupe : BOOL;
	bFilterBlockThisMover : BOOL;
	bStationIsBlocked : BOOL;
	bDummyStation : BOOL; //Station without movers only to change the dynamics of passing movers;
	bTargetFound : BOOL;
	bImTheAsker : BOOL; // Do not return this station as a target
	bStationCanNotBePassed : BOOL;
	
	
	ipActiveStationAStar : I_PathAStarNode;
	ipEmptyPathObj : I_PathAStarNode;
	ipEachPathAhead : I_XP_Path;
	ipPathFoundInOpenList : I_PathAStarNode;
	ipEachAStarNode : I_PathAStarNode;
	ipBesStationAStar : I_PathAStarNode;	
	ipThisStation : I_XP_Station := THIS^;
	
	fPathLength : LREAL;
END_VAR
VAR_INST
	fbLastFoundResult : FB_AStarNode;
END_VAR
VAR_STAT
	fbListNotUsedNodes : FB_CH_List; // Use GetNext() to allways get a not used one
	afbPathAStarNodes : ARRAY[0..(CHALET_BaseComponents.BaseParameterlist.MAX_OBJECTS-1)] OF FB_AStarNode;	
	fbListOpen : FB_CH_List; //To check
	fbListClosed : FB_CH_List; //Allready checked	
END_VAR
//only on first call, add nodes to list of not used objects
IF fbListNotUsedNodes.IsEmpty THEN
	FOR nIdx := 0 TO (CHALET_BaseComponents.BaseParameterlist.MAX_OBJECTS-1) DO
		fbListNotUsedNodes.AddObject(afbPathAStarNodes[nIdx]);
	END_FOR
END_IF

//Clear list
fbListOpen.Clear();
fbListClosed.Clear();

//Init objects in list
fbListNotUsedNodes.ResetIterator();
WHILE fbListNotUsedNodes.HasNextObject() DO
	IF __QUERYINTERFACE(fbListNotUsedNodes.GetNextObject(), ipEachAStarNode) THEN
		IF 	ipEachAStarNode.Station = 0 THEN
			EXIT;//Last used element found, abort
		END_IF
	
		ipEachAStarNode.Station := 0;
		ipEachAStarNode.RouteUsedToNode.Clear();
	END_IF
END_WHILE

//Reset last found result
fbLastFoundResult.Station := 0;
fbLastFoundResult.RouteUsedToNode.Clear();

// Reset once - Use GetNext() to allways get a not used one
fbListNotUsedNodes.ResetIterator();

//This is the start of the search operation. Add this station
__QUERYINTERFACE(fbListNotUsedNodes.GetNextObject(), ipEmptyPathObj);
ipEmptyPathObj.Station := (THIS^);
fbListOpen.AddObject(ipEmptyPathObj);

WHILE NOT fbListOpen.IsEmpty DO
	//Get objet from list with smallest distanse to start-station

	__QUERYINTERFACE(fbListOpen.GetObjectWithLowestNumber(), ipActiveStationAStar);
	//Move objet from open to closed list
	fbListOpen.RemoveObject(ipActiveStationAStar);
	fbListClosed.AddObject(ipActiveStationAStar);
	
	IF ipBesStationAStar <> 0 AND_THEN ipActiveStationAStar.PathLength > ipBesStationAStar.PathLength THEN
		// if a valid station is allreadyx known, skip all station who allready have a larger distance
		CONTINUE;
	END_IF
	
	bImTheAsker := ipActiveStationAStar.Station = ipThisStation;
	bCorrectLUID := (ipActiveStationAStar.Station.LUID = sTargetStation);
 	bCorrectGroupe := (ipActiveStationAStar.Station.TargetGroupe = sTargetStation) OR (sTargetStation =  XPlanarParameterlist.S_ANY_STATION_NAME);
	bDummyStation := (ipActiveStationAStar.Station.MoverQueueSize = 0);//Station without movers only to change the dynamics of passing movers;
	bFilterBlockThisMover := (ipActiveStationAStar.Station.Filter <>  XPlanarParameterlist.S_ANY_STATION_NAME) AND (ipActiveStationAStar.Station.Filter <> sTargetStation) AND NOT bCorrectLUID; // Correct LUID is stronger than filter
	bStationIsBlocked := (ipActiveStationAStar.Station.CtsEmptySpaceInQueue <= 0 AND NOT bDummyStation) OR NOT ipActiveStationAStar.Station.ReadyToRecvMovers;
	bStationCanNotBePassed := ipActiveStationAStar.Station.CtsMoversInQueue > 0 AND NOT bImTheAsker ;
	
	IF (bFilterBlockThisMover OR bStationIsBlocked) AND NOT bImTheAsker THEN
		//Skip
		CONTINUE;
	END_IF
	
	
	IF (bCorrectLUID OR bCorrectGroupe) AND NOT bImTheAsker AND NOT bDummyStation THEN
		//FOUND! - check if way is shorter
		IF ipBesStationAStar=0 OR_ELSE  ipActiveStationAStar.PathLength <= ipBesStationAStar.PathLength THEN
			//shorter - store
			ipBesStationAStar := ipActiveStationAStar;
		END_IF
		
	ELSIF NOT bStationCanNotBePassed THEN		
		// If the destination has not yet been found, set the successor nodes of the current node to the open list
		ipActiveStationAStar.Station.PathsAhead.ResetIterator();
		WHILE ipActiveStationAStar.Station.PathsAhead.HasNextObject() DO
			__QUERYINTERFACE(ipActiveStationAStar.Station.PathsAhead.GetNextObject(), ipEachPathAhead); 
			
